  PROC DrawPart46()
    MoveL Offs(pOrigin,300.79,272.54,0.00),v40,fine,tPen\WObj:=wPaper;
    MoveL Offs(pOrigin,300.79,272.54,6.00),v60,z5,tPen\WObj:=wPaper;
    MoveL Offs(pOrigin,301.42,271.48,6.00),vTravel,z5,tPen\WObj:=wPaper;
    MoveL Offs(pOrigin,301.42,271.48,0.00),v60,z0,tPen\WObj:=wPaper;
    MoveL Offs(pOrigin,301.00,272.11,0.00),v40,z0,tPen\WObj:=wPaper;
    MoveL Offs(pOrigin,301.42,271.48,0.00),v40,z0,tPen\WObj:=wPaper;
    MoveL Offs(pOrigin,301.85,270.62,0.00),v40,z0,tPen\WObj:=wPaper;
    MoveL Offs(pOrigin,301.64,271.05,0.00),v40,z0,tPen\WObj:=wPaper;
    MoveL Offs(pOrigin,301.85,270.62,0.00),v40,fine,tPen\WObj:=wPaper;
    MoveL Offs(pOrigin,301.85,270.62,6.00),v60,z5,tPen\WObj:=wPaper;
    MoveL Offs(pOrigin,295.90,275.73,6.00),vTravel,z5,tPen\WObj:=wPaper;
    MoveL Offs(pOrigin,295.90,275.73,0.00),v60,z0,tPen\WObj:=wPaper;
    MoveL Offs(pOrigin,296.96,276.43,0.00),v40,z0,tPen\WObj:=wPaper;
    MoveL Offs(pOrigin,297.39,277.21,0.00),v40,z0,tPen\WObj:=wPaper;
    MoveL Offs(pOrigin,297.32,277.85,0.00),v40,z0,tPen\WObj:=wPaper;
    MoveL Offs(pOrigin,296.54,278.27,0.00),v40,z0,tPen\WObj:=wPaper;
    MoveL Offs(pOrigin,296.54,278.27,0.00),v40,z0,tPen\WObj:=wPaper;
    MoveL Offs(pOrigin,296.96,280.83,0.00),v40,z0,tPen\WObj:=wPaper;
    MoveL Offs(pOrigin,295.69,281.67,0.00),v40,z0,tPen\WObj:=wPaper;
    MoveL Offs(pOrigin,295.26,281.46,0.00),v40,z0,tPen\WObj:=wPaper;
    MoveL Offs(pOrigin,296.75,284.65,0.00),v40,fine,tPen\WObj:=wPaper;
    MoveL Offs(pOrigin,296.75,284.65,6.00),v60,z5,tPen\WObj:=wPaper;
    MoveL Offs(pOrigin,298.45,283.38,6.00),vTravel,z5,tPen\WObj:=wPaper;
    MoveL Offs(pOrigin,298.45,283.38,0.00),v60,z0,tPen\WObj:=wPaper;
    MoveL Offs(pOrigin,298.02,282.95,0.00),v40,z0,tPen\WObj:=wPaper;
    MoveL Offs(pOrigin,298.02,282.10,0.00),v40,z0,tPen\WObj:=wPaper;
    MoveL Offs(pOrigin,298.45,281.67,0.00),v40,z0,tPen\WObj:=wPaper;
    MoveL Offs(pOrigin,299.09,281.67,0.00),v40,fine,tPen\WObj:=wPaper;
    MoveL Offs(pOrigin,299.09,281.67,6.00),v60,z5,tPen\WObj:=wPaper;
    MoveL Offs(pOrigin,292.71,272.33,6.00),vTravel,z5,tPen\WObj:=wPaper;
    MoveL Offs(pOrigin,292.71,272.33,0.00),v60,z0,tPen\WObj:=wPaper;
    MoveL Offs(pOrigin,293.14,272.75,0.00),v40,z0,tPen\WObj:=wPaper;
    MoveL Offs(pOrigin,292.71,272.33,0.00),v40,fine,tPen\WObj:=wPaper;
    MoveL Offs(pOrigin,292.71,272.33,6.00),v60,z5,tPen\WObj:=wPaper;
    MoveL Offs(pOrigin,291.44,271.48,6.00),vTravel,z5,tPen\WObj:=wPaper;
    MoveL Offs(pOrigin,291.44,271.48,0.00),v60,z0,tPen\WObj:=wPaper;
    MoveL Offs(pOrigin,293.56,273.46,0.00),v40,z0,tPen\WObj:=wPaper;
    MoveL Offs(pOrigin,294.84,274.02,0.00),v40,z0,tPen\WObj:=wPaper;
    MoveL Offs(pOrigin,296.33,274.24,0.00),v40,z0,tPen\WObj:=wPaper;
    MoveL Offs(pOrigin,298.45,273.39,0.00),v40,z0,tPen\WObj:=wPaper;
    MoveL Offs(pOrigin,299.80,271.90,0.00),v40,z0,tPen\WObj:=wPaper;
    MoveL Offs(pOrigin,301.07,269.14,0.00),v40,z0,tPen\WObj:=wPaper;
    MoveL Offs(pOrigin,301.85,266.38,0.00),v40,z0,tPen\WObj:=wPaper;
    MoveL Offs(pOrigin,302.06,264.04,0.00),v40,z0,tPen\WObj:=wPaper;
    MoveL Offs(pOrigin,298.66,250.44,0.00),v40,z0,tPen\WObj:=wPaper;
    MoveL Offs(pOrigin,296.68,240.88,0.00),v40,z0,tPen\WObj:=wPaper;
    MoveL Offs(pOrigin,295.05,239.10,0.00),v40,z0,tPen\WObj:=wPaper;
    MoveL Offs(pOrigin,293.99,238.75,0.00),v40,z0,tPen\WObj:=wPaper;
    MoveL Offs(pOrigin,292.71,239.10,0.00),v40,z0,tPen\WObj:=wPaper;
    MoveL Offs(pOrigin,291.86,240.45,0.00),v40,z0,tPen\WObj:=wPaper;
    MoveL Offs(pOrigin,291.58,243.43,0.00),v40,z0,tPen\WObj:=wPaper;
    MoveL Offs(pOrigin,291.01,243.85,0.00),v40,fine,tPen\WObj:=wPaper;
    MoveL Offs(pOrigin,291.01,243.85,6.00),v60,z5,tPen\WObj:=wPaper;
    MoveL Offs(pOrigin,295.48,239.60,6.00),vTravel,z5,tPen\WObj:=wPaper;
    MoveL Offs(pOrigin,295.48,239.60,0.00),v60,z0,tPen\WObj:=wPaper;
    MoveL Offs(pOrigin,296.11,240.24,0.00),v40,z0,tPen\WObj:=wPaper;
    MoveL Offs(pOrigin,295.48,239.60,0.00),v40,fine,tPen\WObj:=wPaper;
    MoveL Offs(pOrigin,295.48,239.60,6.00),v60,z5,tPen\WObj:=wPaper;
    MoveL Offs(pOrigin,296.33,238.32,6.00),vTravel,z5,tPen\WObj:=wPaper;
    MoveL Offs(pOrigin,296.33,238.32,0.00),v60,z0,tPen\WObj:=wPaper;
    MoveL Offs(pOrigin,296.96,238.96,0.00),v40,z0,tPen\WObj:=wPaper;
    MoveL Offs(pOrigin,296.33,238.32,0.00),v40,fine,tPen\WObj:=wPaper;
    MoveL Offs(pOrigin,296.33,238.32,6.00),v60,z5,tPen\WObj:=wPaper;
    MoveL Offs(pOrigin,297.81,239.39,6.00),vTravel,z5,tPen\WObj:=wPaper;
    MoveL Offs(pOrigin,297.81,239.39,0.00),v60,z0,tPen\WObj:=wPaper;
    MoveL Offs(pOrigin,298.45,239.81,0.00),v40,z0,tPen\WObj:=wPaper;
    MoveL Offs(pOrigin,300.15,239.81,0.00),v40,z0,tPen\WObj:=wPaper;
    MoveL Offs(pOrigin,300.15,239.81,0.00),v40,z0,tPen\WObj:=wPaper;
    MoveL Offs(pOrigin,300.79,240.24,0.00),v40,z0,tPen\WObj:=wPaper;
    MoveL Offs(pOrigin,315.02,240.24,0.00),v40,z0,tPen\WObj:=wPaper;
    MoveL Offs(pOrigin,327.99,239.60,0.00),v40,z0,tPen\WObj:=wPaper;
    MoveL Offs(pOrigin,342.44,238.32,0.00),v40,z0,tPen\WObj:=wPaper;
    MoveL Offs(pOrigin,358.16,235.99,0.00),v40,z0,tPen\WObj:=wPaper;
    MoveL Offs(pOrigin,364.75,234.00,0.00),v40,z0,tPen\WObj:=wPaper;
    MoveL Offs(pOrigin,365.17,233.23,0.00),v40,z0,tPen\WObj:=wPaper;
    MoveL Offs(pOrigin,365.17,233.23,0.00),v40,z0,tPen\WObj:=wPaper;
    MoveL Offs(pOrigin,366.66,232.66,0.00),v40,z0,tPen\WObj:=wPaper;
    MoveL Offs(pOrigin,369.21,230.89,0.00),v40,z0,tPen\WObj:=wPaper;
    MoveL Offs(pOrigin,371.34,228.55,0.00),v40,z0,tPen\WObj:=wPaper;
    MoveL Offs(pOrigin,373.53,224.51,0.00),v40,z0,tPen\WObj:=wPaper;
    MoveL Offs(pOrigin,375.38,218.35,0.00),v40,z0,tPen\WObj:=wPaper;
    MoveL Offs(pOrigin,375.38,218.35,0.00),v40,z0,tPen\WObj:=wPaper;
    MoveL Offs(pOrigin,375.38,217.07,0.00),v40,z0,tPen\WObj:=wPaper;
    MoveL Offs(pOrigin,375.80,216.86,0.00),v40,z0,tPen\WObj:=wPaper;
    MoveL Offs(pOrigin,375.80,216.86,0.00),v40,z0,tPen\WObj:=wPaper;
    MoveL Offs(pOrigin,376.44,217.50,0.00),v40,z0,tPen\WObj:=wPaper;
    MoveL Offs(pOrigin,376.23,218.35,0.00),v40,z0,tPen\WObj:=wPaper;
    MoveL Offs(pOrigin,375.38,218.35,0.00),v40,z0,tPen\WObj:=wPaper;
    MoveL Offs(pOrigin,376.01,218.42,0.00),v40,z0,tPen\WObj:=wPaper;
    MoveL Offs(pOrigin,376.23,218.77,0.00),v40,z0,tPen\WObj:=wPaper;
    MoveL Offs(pOrigin,376.23,222.39,0.00),v40,z0,tPen\WObj:=wPaper;
    MoveL Offs(pOrigin,375.59,226.43,0.00),v40,z0,tPen\WObj:=wPaper;
    MoveL Offs(pOrigin,374.38,230.46,0.00),v40,z0,tPen\WObj:=wPaper;
    MoveL Offs(pOrigin,372.12,234.07,0.00),v40,z0,tPen\WObj:=wPaper;
    MoveL Offs(pOrigin,370.27,235.70,0.00),v40,z0,tPen\WObj:=wPaper;
    MoveL Offs(pOrigin,368.58,236.62,0.00),v40,z0,tPen\WObj:=wPaper;
    MoveL Offs(pOrigin,369.00,236.41,0.00),v40,z0,tPen\WObj:=wPaper;
    MoveL Offs(pOrigin,369.42,236.20,0.00),v40,z0,tPen\WObj:=wPaper;
    MoveL Offs(pOrigin,369.00,236.41,0.00),v40,z0,tPen\WObj:=wPaper;
    MoveL Offs(pOrigin,368.15,236.84,0.00),v40,z0,tPen\WObj:=wPaper;
    MoveL Offs(pOrigin,364.75,238.11,0.00),v40,z0,tPen\WObj:=wPaper;
    MoveL Offs(pOrigin,361.56,238.82,0.00),v40,z0,tPen\WObj:=wPaper;
    MoveL Offs(pOrigin,361.14,239.39,0.00),v40,fine,tPen\WObj:=wPaper;
    MoveL Offs(pOrigin,361.14,239.39,6.00),v60,z5,tPen\WObj:=wPaper;
    MoveL Offs(pOrigin,357.52,239.60,6.00),vTravel,z5,tPen\WObj:=wPaper;
    MoveL Offs(pOrigin,357.52,239.60,0.00),v60,z0,tPen\WObj:=wPaper;
    MoveL Offs(pOrigin,364.75,239.39,0.00),v40,z0,tPen\WObj:=wPaper;
    MoveL Offs(pOrigin,369.21,237.97,0.00),v40,z0,tPen\WObj:=wPaper;
    MoveL Offs(pOrigin,371.55,236.62,0.00),v40,z0,tPen\WObj:=wPaper;
    MoveL Offs(pOrigin,373.25,235.14,0.00),v40,z0,tPen\WObj:=wPaper;
    MoveL Offs(pOrigin,374.81,233.01,0.00),v40,z0,tPen\WObj:=wPaper;
    MoveL Offs(pOrigin,375.87,230.68,0.00),v40,z0,tPen\WObj:=wPaper;
    MoveL Offs(pOrigin,377.08,226.64,0.00),v40,z0,tPen\WObj:=wPaper;
    MoveL Offs(pOrigin,377.71,221.96,0.00),v40,z0,tPen\WObj:=wPaper;
    MoveL Offs(pOrigin,377.71,212.82,0.00),v40,z0,tPen\WObj:=wPaper;
    MoveL Offs(pOrigin,376.86,204.96,0.00),v40,z0,tPen\WObj:=wPaper;
    MoveL Offs(pOrigin,373.89,190.51,0.00),v40,z0,tPen\WObj:=wPaper;
    MoveL Offs(pOrigin,376.23,188.60,0.00),v40,z0,tPen\WObj:=wPaper;
    MoveL Offs(pOrigin,377.92,186.48,0.00),v40,z0,tPen\WObj:=wPaper;
    MoveL Offs(pOrigin,378.35,186.90,0.00),v40,z0,tPen\WObj:=wPaper;
  ENDPROC

  PROC DrawPart47()
    MoveL Offs(pOrigin,380.26,204.75,0.00),v40,z0,tPen\WObj:=wPaper;
    MoveL Offs(pOrigin,380.48,217.93,0.00),v40,z0,tPen\WObj:=wPaper;
    MoveL Offs(pOrigin,379.62,225.79,0.00),v40,z0,tPen\WObj:=wPaper;
    MoveL Offs(pOrigin,378.99,228.55,0.00),v40,z0,tPen\WObj:=wPaper;
    MoveL Offs(pOrigin,377.50,232.59,0.00),v40,z0,tPen\WObj:=wPaper;
    MoveL Offs(pOrigin,377.50,233.44,0.00),v40,z0,tPen\WObj:=wPaper;
    MoveL Offs(pOrigin,377.50,233.44,0.00),v40,z0,tPen\WObj:=wPaper;
    MoveL Offs(pOrigin,378.35,233.30,0.00),v40,z0,tPen\WObj:=wPaper;
    MoveL Offs(pOrigin,379.41,231.52,0.00),v40,z0,tPen\WObj:=wPaper;
    MoveL Offs(pOrigin,379.41,231.52,0.00),v40,z0,tPen\WObj:=wPaper;
    MoveL Offs(pOrigin,380.33,231.10,0.00),v40,z0,tPen\WObj:=wPaper;
    MoveL Offs(pOrigin,381.61,228.55,0.00),v40,z0,tPen\WObj:=wPaper;
    MoveL Offs(pOrigin,383.45,222.39,0.00),v40,z0,tPen\WObj:=wPaper;
    MoveL Offs(pOrigin,384.30,217.50,0.00),v40,z0,tPen\WObj:=wPaper;
    MoveL Offs(pOrigin,388.55,169.69,0.00),v40,z0,tPen\WObj:=wPaper;
    MoveL Offs(pOrigin,392.80,129.31,0.00),v40,z0,tPen\WObj:=wPaper;
    MoveL Offs(pOrigin,392.59,128.46,0.00),v40,z0,tPen\WObj:=wPaper;
    MoveL Offs(pOrigin,391.60,128.68,0.00),v40,z0,tPen\WObj:=wPaper;
    MoveL Offs(pOrigin,391.10,129.95,0.00),v40,z0,tPen\WObj:=wPaper;
    MoveL Offs(pOrigin,390.46,139.30,0.00),v40,z0,tPen\WObj:=wPaper;
    MoveL Offs(pOrigin,389.54,141.43,0.00),v40,z0,tPen\WObj:=wPaper;
    MoveL Offs(pOrigin,387.13,143.76,0.00),v40,z0,tPen\WObj:=wPaper;
    MoveL Offs(pOrigin,386.85,144.61,0.00),v40,z0,tPen\WObj:=wPaper;
    MoveL Offs(pOrigin,387.27,147.16,0.00),v40,z0,tPen\WObj:=wPaper;
    MoveL Offs(pOrigin,387.06,149.71,0.00),v40,z0,tPen\WObj:=wPaper;
    MoveL Offs(pOrigin,385.01,155.02,0.00),v40,z0,tPen\WObj:=wPaper;
    MoveL Offs(pOrigin,382.53,159.91,0.00),v40,z0,tPen\WObj:=wPaper;
    MoveL Offs(pOrigin,380.90,164.80,0.00),v40,z0,tPen\WObj:=wPaper;
    MoveL Offs(pOrigin,380.90,166.93,0.00),v40,z0,tPen\WObj:=wPaper;
    MoveL Offs(pOrigin,381.75,169.26,0.00),v40,z0,tPen\WObj:=wPaper;
    MoveL Offs(pOrigin,381.75,171.39,0.00),v40,z0,tPen\WObj:=wPaper;
    MoveL Offs(pOrigin,379.20,179.25,0.00),v40,z0,tPen\WObj:=wPaper;
    MoveL Offs(pOrigin,378.56,182.65,0.00),v40,z0,tPen\WObj:=wPaper;
    MoveL Offs(pOrigin,378.77,185.62,0.00),v40,z0,tPen\WObj:=wPaper;
    MoveL Offs(pOrigin,378.77,185.62,0.00),v40,z0,tPen\WObj:=wPaper;
    MoveL Offs(pOrigin,377.92,185.84,0.00),v40,z0,tPen\WObj:=wPaper;
    MoveL Offs(pOrigin,378.35,186.90,0.00),v40,z0,tPen\WObj:=wPaper;
    MoveL Offs(pOrigin,378.99,186.90,0.00),v40,z0,tPen\WObj:=wPaper;
    MoveL Offs(pOrigin,381.11,199.86,0.00),v40,z0,tPen\WObj:=wPaper;
    MoveL Offs(pOrigin,381.96,211.12,0.00),v40,z0,tPen\WObj:=wPaper;
    MoveL Offs(pOrigin,381.54,221.96,0.00),v40,z0,tPen\WObj:=wPaper;
    MoveL Offs(pOrigin,381.11,224.94,0.00),v40,z0,tPen\WObj:=wPaper;
    MoveL Offs(pOrigin,379.41,230.68,0.00),v40,z0,tPen\WObj:=wPaper;
    MoveL Offs(pOrigin,379.41,231.52,0.00),v40,fine,tPen\WObj:=wPaper;
    MoveL Offs(pOrigin,379.41,231.52,6.00),v60,z5,tPen\WObj:=wPaper;
    MoveL Offs(pOrigin,380.48,230.46,6.00),vTravel,z5,tPen\WObj:=wPaper;
    MoveL Offs(pOrigin,380.48,230.46,0.00),v60,z0,tPen\WObj:=wPaper;
    MoveL Offs(pOrigin,380.26,230.89,0.00),v40,z0,tPen\WObj:=wPaper;
    MoveL Offs(pOrigin,380.48,230.46,0.00),v40,fine,tPen\WObj:=wPaper;
    MoveL Offs(pOrigin,380.48,230.46,6.00),v60,z5,tPen\WObj:=wPaper;
    MoveL Offs(pOrigin,381.75,231.52,6.00),vTravel,z5,tPen\WObj:=wPaper;
    MoveL Offs(pOrigin,381.75,231.52,0.00),v60,z0,tPen\WObj:=wPaper;
    MoveL Offs(pOrigin,381.54,231.95,0.00),v40,z0,tPen\WObj:=wPaper;
    MoveL Offs(pOrigin,381.75,231.52,0.00),v40,fine,tPen\WObj:=wPaper;
    MoveL Offs(pOrigin,381.75,231.52,6.00),v60,z5,tPen\WObj:=wPaper;
    MoveL Offs(pOrigin,380.69,233.23,6.00),vTravel,z5,tPen\WObj:=wPaper;
    MoveL Offs(pOrigin,380.69,233.23,0.00),v60,z0,tPen\WObj:=wPaper;
    MoveL Offs(pOrigin,380.26,233.86,0.00),v40,z0,tPen\WObj:=wPaper;
    MoveL Offs(pOrigin,380.69,233.23,0.00),v40,fine,tPen\WObj:=wPaper;
    MoveL Offs(pOrigin,380.69,233.23,6.00),v60,z5,tPen\WObj:=wPaper;
    MoveL Offs(pOrigin,379.84,234.29,6.00),vTravel,z5,tPen\WObj:=wPaper;
    MoveL Offs(pOrigin,379.84,234.29,0.00),v60,z0,tPen\WObj:=wPaper;
    MoveL Offs(pOrigin,379.41,234.93,0.00),v40,z0,tPen\WObj:=wPaper;
    MoveL Offs(pOrigin,379.84,234.29,0.00),v40,z0,tPen\WObj:=wPaper;
    MoveL Offs(pOrigin,379.20,235.14,0.00),v40,z0,tPen\WObj:=wPaper;
    MoveL Offs(pOrigin,377.71,236.62,0.00),v40,z0,tPen\WObj:=wPaper;
    MoveL Offs(pOrigin,379.20,235.14,0.00),v40,fine,tPen\WObj:=wPaper;
    MoveL Offs(pOrigin,379.20,235.14,6.00),v60,z5,tPen\WObj:=wPaper;
    MoveL Offs(pOrigin,377.50,233.44,6.00),vTravel,z5,tPen\WObj:=wPaper;
    MoveL Offs(pOrigin,377.50,233.44,0.00),v60,z0,tPen\WObj:=wPaper;
    MoveL Offs(pOrigin,377.08,234.50,0.00),v40,z0,tPen\WObj:=wPaper;
    MoveL Offs(pOrigin,375.66,235.42,0.00),v40,z0,tPen\WObj:=wPaper;
    MoveL Offs(pOrigin,373.46,237.69,0.00),v40,z0,tPen\WObj:=wPaper;
    MoveL Offs(pOrigin,373.04,237.90,0.00),v40,z0,tPen\WObj:=wPaper;
    MoveL Offs(pOrigin,369.42,239.39,0.00),v40,z0,tPen\WObj:=wPaper;
    MoveL Offs(pOrigin,364.54,240.66,0.00),v40,z0,tPen\WObj:=wPaper;
    MoveL Offs(pOrigin,356.89,241.94,0.00),v40,z0,tPen\WObj:=wPaper;
    MoveL Offs(pOrigin,341.38,243.64,0.00),v40,z0,tPen\WObj:=wPaper;
    MoveL Offs(pOrigin,320.55,244.91,0.00),v40,z0,tPen\WObj:=wPaper;
    MoveL Offs(pOrigin,302.06,245.12,0.00),v40,z0,tPen\WObj:=wPaper;
    MoveL Offs(pOrigin,299.30,244.91,0.00),v40,z0,tPen\WObj:=wPaper;
    MoveL Offs(pOrigin,298.88,244.27,0.00),v40,z0,tPen\WObj:=wPaper;
    MoveL Offs(pOrigin,297.88,240.24,0.00),v40,z0,tPen\WObj:=wPaper;
    MoveL Offs(pOrigin,298.02,239.81,0.00),v40,z0,tPen\WObj:=wPaper;
    MoveL Offs(pOrigin,298.02,239.81,0.00),v40,z0,tPen\WObj:=wPaper;
    MoveL Offs(pOrigin,295.26,237.83,0.00),v40,z0,tPen\WObj:=wPaper;
    MoveL Offs(pOrigin,294.20,237.48,0.00),v40,z0,tPen\WObj:=wPaper;
    MoveL Offs(pOrigin,291.93,237.69,0.00),v40,z0,tPen\WObj:=wPaper;
    MoveL Offs(pOrigin,291.44,233.44,0.00),v40,z0,tPen\WObj:=wPaper;
    MoveL Offs(pOrigin,289.24,226.43,0.00),v40,z0,tPen\WObj:=wPaper;
    MoveL Offs(pOrigin,295.97,218.35,0.00),v40,z0,tPen\WObj:=wPaper;
    MoveL Offs(pOrigin,300.79,213.75,0.00),v40,z0,tPen\WObj:=wPaper;
    MoveL Offs(pOrigin,310.14,211.34,0.00),v40,z0,tPen\WObj:=wPaper;
    MoveL Offs(pOrigin,317.58,208.86,0.00),v40,z0,tPen\WObj:=wPaper;
    MoveL Offs(pOrigin,336.27,201.07,0.00),v40,z0,tPen\WObj:=wPaper;
    MoveL Offs(pOrigin,346.90,197.52,0.00),v40,z0,tPen\WObj:=wPaper;
    MoveL Offs(pOrigin,366.88,192.21,0.00),v40,z0,tPen\WObj:=wPaper;
    MoveL Offs(pOrigin,371.76,190.51,0.00),v40,z0,tPen\WObj:=wPaper;
    MoveL Offs(pOrigin,372.33,190.58,0.00),v40,z0,tPen\WObj:=wPaper;
    MoveL Offs(pOrigin,373.89,196.89,0.00),v40,z0,tPen\WObj:=wPaper;
    MoveL Offs(pOrigin,375.38,205.18,0.00),v40,z0,tPen\WObj:=wPaper;
    MoveL Offs(pOrigin,375.80,208.79,0.00),v40,z0,tPen\WObj:=wPaper;
    MoveL Offs(pOrigin,375.80,216.86,0.00),v40,fine,tPen\WObj:=wPaper;
    MoveL Offs(pOrigin,375.80,216.86,6.00),v60,z5,tPen\WObj:=wPaper;
    MoveL Offs(pOrigin,371.98,227.27,6.00),vTravel,z5,tPen\WObj:=wPaper;
    MoveL Offs(pOrigin,371.98,227.27,0.00),v60,z0,tPen\WObj:=wPaper;
    MoveL Offs(pOrigin,371.55,227.91,0.00),v40,z0,tPen\WObj:=wPaper;
    MoveL Offs(pOrigin,371.98,227.27,0.00),v40,fine,tPen\WObj:=wPaper;
    MoveL Offs(pOrigin,371.98,227.27,6.00),v60,z5,tPen\WObj:=wPaper;
    MoveL Offs(pOrigin,370.49,229.40,6.00),vTravel,z5,tPen\WObj:=wPaper;
    MoveL Offs(pOrigin,370.49,229.40,0.00),v60,z0,tPen\WObj:=wPaper;
    MoveL Offs(pOrigin,369.85,230.04,0.00),v40,z0,tPen\WObj:=wPaper;
    MoveL Offs(pOrigin,370.49,229.40,0.00),v40,fine,tPen\WObj:=wPaper;
    MoveL Offs(pOrigin,370.49,229.40,6.00),v60,z5,tPen\WObj:=wPaper;
    MoveL Offs(pOrigin,369.64,230.25,6.00),vTravel,z5,tPen\WObj:=wPaper;
    MoveL Offs(pOrigin,369.64,230.25,0.00),v60,z0,tPen\WObj:=wPaper;
    MoveL Offs(pOrigin,369.00,230.89,0.00),v40,z0,tPen\WObj:=wPaper;
    MoveL Offs(pOrigin,369.64,230.25,0.00),v40,fine,tPen\WObj:=wPaper;
    MoveL Offs(pOrigin,369.64,230.25,6.00),v60,z5,tPen\WObj:=wPaper;
    MoveL Offs(pOrigin,373.46,231.95,6.00),vTravel,z5,tPen\WObj:=wPaper;
  ENDPROC

  PROC DrawPart48()
    MoveL Offs(pOrigin,373.46,231.95,0.00),v60,z0,tPen\WObj:=wPaper;
    MoveL Offs(pOrigin,373.25,232.38,0.00),v40,z0,tPen\WObj:=wPaper;
    MoveL Offs(pOrigin,373.46,231.95,0.00),v40,fine,tPen\WObj:=wPaper;
    MoveL Offs(pOrigin,373.46,231.95,6.00),v60,z5,tPen\WObj:=wPaper;
    MoveL Offs(pOrigin,374.10,230.68,6.00),vTravel,z5,tPen\WObj:=wPaper;
    MoveL Offs(pOrigin,374.10,230.68,0.00),v60,z0,tPen\WObj:=wPaper;
    MoveL Offs(pOrigin,373.89,231.10,0.00),v40,z0,tPen\WObj:=wPaper;
    MoveL Offs(pOrigin,374.10,230.68,0.00),v40,fine,tPen\WObj:=wPaper;
    MoveL Offs(pOrigin,374.10,230.68,6.00),v60,z5,tPen\WObj:=wPaper;
    MoveL Offs(pOrigin,375.16,231.95,6.00),vTravel,z5,tPen\WObj:=wPaper;
    MoveL Offs(pOrigin,375.16,231.95,0.00),v60,z0,tPen\WObj:=wPaper;
    MoveL Offs(pOrigin,374.95,232.38,0.00),v40,z0,tPen\WObj:=wPaper;
    MoveL Offs(pOrigin,375.16,231.95,0.00),v40,z0,tPen\WObj:=wPaper;
    MoveL Offs(pOrigin,374.74,232.80,0.00),v40,z0,tPen\WObj:=wPaper;
    MoveL Offs(pOrigin,374.31,233.44,0.00),v40,z0,tPen\WObj:=wPaper;
    MoveL Offs(pOrigin,374.74,232.80,0.00),v40,fine,tPen\WObj:=wPaper;
    MoveL Offs(pOrigin,374.74,232.80,6.00),v60,z5,tPen\WObj:=wPaper;
    MoveL Offs(pOrigin,374.10,233.86,6.00),vTravel,z5,tPen\WObj:=wPaper;
    MoveL Offs(pOrigin,374.10,233.86,0.00),v60,z0,tPen\WObj:=wPaper;
    MoveL Offs(pOrigin,373.46,234.50,0.00),v40,z0,tPen\WObj:=wPaper;
    MoveL Offs(pOrigin,374.10,233.86,0.00),v40,fine,tPen\WObj:=wPaper;
    MoveL Offs(pOrigin,374.10,233.86,6.00),v60,z5,tPen\WObj:=wPaper;
    MoveL Offs(pOrigin,373.25,234.93,6.00),vTravel,z5,tPen\WObj:=wPaper;
    MoveL Offs(pOrigin,373.25,234.93,0.00),v60,z0,tPen\WObj:=wPaper;
    MoveL Offs(pOrigin,372.40,235.77,0.00),v40,z0,tPen\WObj:=wPaper;
    MoveL Offs(pOrigin,373.25,234.93,0.00),v40,fine,tPen\WObj:=wPaper;
    MoveL Offs(pOrigin,373.25,234.93,6.00),v60,z5,tPen\WObj:=wPaper;
    MoveL Offs(pOrigin,372.61,233.44,6.00),vTravel,z5,tPen\WObj:=wPaper;
    MoveL Offs(pOrigin,372.61,233.44,0.00),v60,z0,tPen\WObj:=wPaper;
    MoveL Offs(pOrigin,372.83,233.01,0.00),v40,z0,tPen\WObj:=wPaper;
    MoveL Offs(pOrigin,372.61,233.44,0.00),v40,z0,tPen\WObj:=wPaper;
    MoveL Offs(pOrigin,372.19,233.65,0.00),v40,z0,tPen\WObj:=wPaper;
    MoveL Offs(pOrigin,371.98,234.07,0.00),v40,z0,tPen\WObj:=wPaper;
    MoveL Offs(pOrigin,372.19,233.65,0.00),v40,fine,tPen\WObj:=wPaper;
    MoveL Offs(pOrigin,372.19,233.65,6.00),v60,z5,tPen\WObj:=wPaper;
    MoveL Offs(pOrigin,370.70,235.35,6.00),vTravel,z5,tPen\WObj:=wPaper;
    MoveL Offs(pOrigin,370.70,235.35,0.00),v60,z0,tPen\WObj:=wPaper;
    MoveL Offs(pOrigin,371.12,235.14,0.00),v40,z0,tPen\WObj:=wPaper;
    MoveL Offs(pOrigin,370.70,235.35,0.00),v40,z0,tPen\WObj:=wPaper;
    MoveL Offs(pOrigin,369.85,235.99,0.00),v40,z0,tPen\WObj:=wPaper;
    MoveL Offs(pOrigin,370.27,235.56,0.00),v40,z0,tPen\WObj:=wPaper;
    MoveL Offs(pOrigin,369.85,235.99,0.00),v40,fine,tPen\WObj:=wPaper;
    MoveL Offs(pOrigin,369.85,235.99,6.00),v60,z5,tPen\WObj:=wPaper;
    MoveL Offs(pOrigin,371.76,236.20,6.00),vTravel,z5,tPen\WObj:=wPaper;
    MoveL Offs(pOrigin,371.76,236.20,0.00),v60,z0,tPen\WObj:=wPaper;
    MoveL Offs(pOrigin,371.34,236.62,0.00),v40,z0,tPen\WObj:=wPaper;
    MoveL Offs(pOrigin,371.76,236.20,0.00),v40,fine,tPen\WObj:=wPaper;
    MoveL Offs(pOrigin,371.76,236.20,6.00),v60,z5,tPen\WObj:=wPaper;
    MoveL Offs(pOrigin,373.89,237.48,6.00),vTravel,z5,tPen\WObj:=wPaper;
    MoveL Offs(pOrigin,373.89,237.48,0.00),v60,z0,tPen\WObj:=wPaper;
    MoveL Offs(pOrigin,374.10,237.05,0.00),v40,z0,tPen\WObj:=wPaper;
    MoveL Offs(pOrigin,373.89,237.48,0.00),v40,z0,tPen\WObj:=wPaper;
    MoveL Offs(pOrigin,374.52,236.84,0.00),v40,z0,tPen\WObj:=wPaper;
    MoveL Offs(pOrigin,374.74,236.41,0.00),v40,z0,tPen\WObj:=wPaper;
    MoveL Offs(pOrigin,374.52,236.84,0.00),v40,z0,tPen\WObj:=wPaper;
    MoveL Offs(pOrigin,375.16,236.20,0.00),v40,z0,tPen\WObj:=wPaper;
    MoveL Offs(pOrigin,375.38,235.77,0.00),v40,z0,tPen\WObj:=wPaper;
    MoveL Offs(pOrigin,375.16,236.20,0.00),v40,fine,tPen\WObj:=wPaper;
    MoveL Offs(pOrigin,375.16,236.20,6.00),v60,z5,tPen\WObj:=wPaper;
    MoveL Offs(pOrigin,365.17,233.23,6.00),vTravel,z5,tPen\WObj:=wPaper;
    MoveL Offs(pOrigin,365.17,233.23,0.00),v60,z0,tPen\WObj:=wPaper;
    MoveL Offs(pOrigin,356.46,235.35,0.00),v40,z0,tPen\WObj:=wPaper;
    MoveL Offs(pOrigin,339.89,237.48,0.00),v40,z0,tPen\WObj:=wPaper;
    MoveL Offs(pOrigin,320.12,238.96,0.00),v40,z0,tPen\WObj:=wPaper;
    MoveL Offs(pOrigin,300.58,239.39,0.00),v40,z0,tPen\WObj:=wPaper;
    MoveL Offs(pOrigin,300.15,239.81,0.00),v40,fine,tPen\WObj:=wPaper;
    MoveL Offs(pOrigin,300.15,239.81,6.00),v60,z5,tPen\WObj:=wPaper;
    MoveL Offs(pOrigin,289.52,226.21,6.00),vTravel,z5,tPen\WObj:=wPaper;
    MoveL Offs(pOrigin,289.52,226.21,0.00),v60,z0,tPen\WObj:=wPaper;
    MoveL Offs(pOrigin,289.74,225.79,0.00),v40,z0,tPen\WObj:=wPaper;
    MoveL Offs(pOrigin,289.52,226.21,0.00),v40,fine,tPen\WObj:=wPaper;
    MoveL Offs(pOrigin,289.52,226.21,6.00),v60,z5,tPen\WObj:=wPaper;
    MoveL Offs(pOrigin,290.59,224.94,6.00),vTravel,z5,tPen\WObj:=wPaper;
    MoveL Offs(pOrigin,290.59,224.94,0.00),v60,z0,tPen\WObj:=wPaper;
    MoveL Offs(pOrigin,290.80,224.51,0.00),v40,z0,tPen\WObj:=wPaper;
    MoveL Offs(pOrigin,290.59,224.94,0.00),v40,fine,tPen\WObj:=wPaper;
    MoveL Offs(pOrigin,290.59,224.94,6.00),v60,z5,tPen\WObj:=wPaper;
    MoveL Offs(pOrigin,289.52,223.24,6.00),vTravel,z5,tPen\WObj:=wPaper;
    MoveL Offs(pOrigin,289.52,223.24,0.00),v60,z0,tPen\WObj:=wPaper;
    MoveL Offs(pOrigin,290.80,222.60,0.00),v40,z0,tPen\WObj:=wPaper;
    MoveL Offs(pOrigin,294.20,218.35,0.00),v40,z0,tPen\WObj:=wPaper;
    MoveL Offs(pOrigin,301.21,211.34,0.00),v40,z0,tPen\WObj:=wPaper;
    MoveL Offs(pOrigin,313.75,195.61,0.00),v40,z0,tPen\WObj:=wPaper;
    MoveL Offs(pOrigin,313.68,194.76,0.00),v40,z0,tPen\WObj:=wPaper;
    MoveL Offs(pOrigin,302.06,189.24,0.00),v40,z0,tPen\WObj:=wPaper;
    MoveL Offs(pOrigin,300.79,189.38,0.00),v40,z0,tPen\WObj:=wPaper;
    MoveL Offs(pOrigin,297.81,191.22,0.00),v40,z0,tPen\WObj:=wPaper;
    MoveL Offs(pOrigin,297.32,190.94,0.00),v40,z0,tPen\WObj:=wPaper;
    MoveL Offs(pOrigin,297.39,190.51,0.00),v40,z0,tPen\WObj:=wPaper;
    MoveL Offs(pOrigin,302.27,187.47,0.00),v40,z0,tPen\WObj:=wPaper;
    MoveL Offs(pOrigin,316.94,182.23,0.00),v40,z0,tPen\WObj:=wPaper;
    MoveL Offs(pOrigin,317.15,181.59,0.00),v40,z0,tPen\WObj:=wPaper;
    MoveL Offs(pOrigin,309.71,159.27,0.00),v40,z0,tPen\WObj:=wPaper;
    MoveL Offs(pOrigin,291.65,101.26,0.00),v40,z0,tPen\WObj:=wPaper;
    MoveL Offs(pOrigin,286.98,81.71,0.00),v40,z0,tPen\WObj:=wPaper;
    MoveL Offs(pOrigin,285.49,73.21,0.00),v40,z0,tPen\WObj:=wPaper;
    MoveL Offs(pOrigin,285.06,68.75,0.00),v40,z0,tPen\WObj:=wPaper;
    MoveL Offs(pOrigin,281.88,68.54,0.00),v40,z0,tPen\WObj:=wPaper;
    MoveL Offs(pOrigin,276.14,66.62,0.00),v40,z0,tPen\WObj:=wPaper;
    MoveL Offs(pOrigin,275.50,68.54,0.00),v40,z0,tPen\WObj:=wPaper;
    MoveL Offs(pOrigin,273.59,80.44,0.00),v40,z0,tPen\WObj:=wPaper;
    MoveL Offs(pOrigin,272.31,92.97,0.00),v40,z0,tPen\WObj:=wPaper;
    MoveL Offs(pOrigin,271.89,100.41,0.00),v40,z0,tPen\WObj:=wPaper;
    MoveL Offs(pOrigin,271.89,111.68,0.00),v40,z0,tPen\WObj:=wPaper;
    MoveL Offs(pOrigin,272.52,122.30,0.00),v40,z0,tPen\WObj:=wPaper;
    MoveL Offs(pOrigin,274.23,137.18,0.00),v40,z0,tPen\WObj:=wPaper;
    MoveL Offs(pOrigin,277.62,157.57,0.00),v40,z0,tPen\WObj:=wPaper;
    MoveL Offs(pOrigin,281.45,175.64,0.00),v40,z0,tPen\WObj:=wPaper;
    MoveL Offs(pOrigin,286.98,197.74,0.00),v40,z0,tPen\WObj:=wPaper;
    MoveL Offs(pOrigin,287.61,198.59,0.00),v40,fine,tPen\WObj:=wPaper;
    MoveL Offs(pOrigin,287.61,198.59,6.00),v60,z5,tPen\WObj:=wPaper;
    MoveL Offs(pOrigin,293.35,194.34,6.00),vTravel,z5,tPen\WObj:=wPaper;
    MoveL Offs(pOrigin,293.35,194.34,0.00),v60,z0,tPen\WObj:=wPaper;
    MoveL Offs(pOrigin,287.40,199.23,0.00),v40,z0,tPen\WObj:=wPaper;
    MoveL Offs(pOrigin,289.74,212.19,0.00),v40,z0,tPen\WObj:=wPaper;
    MoveL Offs(pOrigin,289.95,218.14,0.00),v40,z0,tPen\WObj:=wPaper;
    MoveL Offs(pOrigin,289.52,223.24,0.00),v40,fine,tPen\WObj:=wPaper;
    MoveL Offs(pOrigin,289.52,223.24,6.00),v60,z5,tPen\WObj:=wPaper;
    MoveL Offs(pOrigin,288.25,222.18,6.00),vTravel,z5,tPen\WObj:=wPaper;
    MoveL Offs(pOrigin,288.25,222.18,0.00),v60,z0,tPen\WObj:=wPaper;
  ENDPROC

  PROC DrawPart49()
    MoveL Offs(pOrigin,288.18,221.11,0.00),v40,z0,tPen\WObj:=wPaper;
    MoveL Offs(pOrigin,287.75,220.69,0.00),v40,z0,tPen\WObj:=wPaper;
    MoveL Offs(pOrigin,285.77,215.38,0.00),v40,z0,tPen\WObj:=wPaper;
    MoveL Offs(pOrigin,280.88,205.39,0.00),v40,z0,tPen\WObj:=wPaper;
    MoveL Offs(pOrigin,274.93,195.19,0.00),v40,z0,tPen\WObj:=wPaper;
    MoveL Offs(pOrigin,261.55,175.21,0.00),v40,z0,tPen\WObj:=wPaper;
    MoveL Offs(pOrigin,260.62,171.39,0.00),v40,z0,tPen\WObj:=wPaper;
    MoveL Offs(pOrigin,259.63,169.05,0.00),v40,z0,tPen\WObj:=wPaper;
    MoveL Offs(pOrigin,257.65,166.71,0.00),v40,z0,tPen\WObj:=wPaper;
    MoveL Offs(pOrigin,252.55,162.25,0.00),v40,z0,tPen\WObj:=wPaper;
    MoveL Offs(pOrigin,250.00,159.49,0.00),v40,z0,tPen\WObj:=wPaper;
    MoveL Offs(pOrigin,247.73,156.51,0.00),v40,z0,tPen\WObj:=wPaper;
    MoveL Offs(pOrigin,246.60,152.69,0.00),v40,z0,tPen\WObj:=wPaper;
    MoveL Offs(pOrigin,245.96,152.69,0.00),v40,z0,tPen\WObj:=wPaper;
    MoveL Offs(pOrigin,247.52,157.36,0.00),v40,z0,tPen\WObj:=wPaper;
    MoveL Offs(pOrigin,249.36,160.12,0.00),v40,z0,tPen\WObj:=wPaper;
    MoveL Offs(pOrigin,251.70,162.68,0.00),v40,z0,tPen\WObj:=wPaper;
    MoveL Offs(pOrigin,251.91,163.95,0.00),v40,z0,tPen\WObj:=wPaper;
    MoveL Offs(pOrigin,245.11,169.48,0.00),v40,z0,tPen\WObj:=wPaper;
    MoveL Offs(pOrigin,243.98,171.60,0.00),v40,z0,tPen\WObj:=wPaper;
    MoveL Offs(pOrigin,241.36,179.25,0.00),v40,z0,tPen\WObj:=wPaper;
    MoveL Offs(pOrigin,239.23,183.29,0.00),v40,z0,tPen\WObj:=wPaper;
    MoveL Offs(pOrigin,230.80,195.40,0.00),v40,z0,tPen\WObj:=wPaper;
    MoveL Offs(pOrigin,224.93,205.39,0.00),v40,z0,tPen\WObj:=wPaper;
    MoveL Offs(pOrigin,222.16,208.15,0.00),v40,z0,tPen\WObj:=wPaper;
    MoveL Offs(pOrigin,221.31,208.57,0.00),v40,z0,tPen\WObj:=wPaper;
    MoveL Offs(pOrigin,221.10,207.30,0.00),v40,z0,tPen\WObj:=wPaper;
    MoveL Offs(pOrigin,222.16,201.14,0.00),v40,z0,tPen\WObj:=wPaper;
    MoveL Offs(pOrigin,224.93,189.24,0.00),v40,z0,tPen\WObj:=wPaper;
    MoveL Offs(pOrigin,227.05,178.40,0.00),v40,z0,tPen\WObj:=wPaper;
    MoveL Offs(pOrigin,227.26,175.85,0.00),v40,z0,tPen\WObj:=wPaper;
    MoveL Offs(pOrigin,227.69,175.21,0.00),v40,z0,tPen\WObj:=wPaper;
    MoveL Offs(pOrigin,227.69,175.21,0.00),v40,z0,tPen\WObj:=wPaper;
    MoveL Offs(pOrigin,228.04,175.43,0.00),v40,z0,tPen\WObj:=wPaper;
    MoveL Offs(pOrigin,228.32,176.49,0.00),v40,z0,tPen\WObj:=wPaper;
    MoveL Offs(pOrigin,228.75,183.71,0.00),v40,z0,tPen\WObj:=wPaper;
    MoveL Offs(pOrigin,229.53,186.48,0.00),v40,z0,tPen\WObj:=wPaper;
    MoveL Offs(pOrigin,230.66,187.75,0.00),v40,z0,tPen\WObj:=wPaper;
    MoveL Offs(pOrigin,231.94,188.39,0.00),v40,z0,tPen\WObj:=wPaper;
    MoveL Offs(pOrigin,233.57,188.10,0.00),v40,z0,tPen\WObj:=wPaper;
    MoveL Offs(pOrigin,233.85,187.32,0.00),v40,z0,tPen\WObj:=wPaper;
    MoveL Offs(pOrigin,233.85,187.32,0.00),v40,z0,tPen\WObj:=wPaper;
    MoveL Offs(pOrigin,236.19,184.99,0.00),v40,z0,tPen\WObj:=wPaper;
    MoveL Offs(pOrigin,237.18,183.50,0.00),v40,z0,tPen\WObj:=wPaper;
    MoveL Offs(pOrigin,237.46,182.23,0.00),v40,z0,tPen\WObj:=wPaper;
    MoveL Offs(pOrigin,237.46,182.23,0.00),v40,z0,tPen\WObj:=wPaper;
    MoveL Offs(pOrigin,238.95,179.25,0.00),v40,z0,tPen\WObj:=wPaper;
    MoveL Offs(pOrigin,238.88,177.55,0.00),v40,z0,tPen\WObj:=wPaper;
    MoveL Offs(pOrigin,238.10,176.91,0.00),v40,z0,tPen\WObj:=wPaper;
    MoveL Offs(pOrigin,237.04,177.05,0.00),v40,z0,tPen\WObj:=wPaper;
    MoveL Offs(pOrigin,236.19,177.76,0.00),v40,z0,tPen\WObj:=wPaper;
    MoveL Offs(pOrigin,235.98,178.61,0.00),v40,z0,tPen\WObj:=wPaper;
    MoveL Offs(pOrigin,235.98,178.61,0.00),v40,z0,tPen\WObj:=wPaper;
    MoveL Offs(pOrigin,235.48,179.04,0.00),v40,z0,tPen\WObj:=wPaper;
    MoveL Offs(pOrigin,235.12,180.10,0.00),v40,z0,tPen\WObj:=wPaper;
    MoveL Offs(pOrigin,235.27,181.59,0.00),v40,z0,tPen\WObj:=wPaper;
    MoveL Offs(pOrigin,236.19,182.23,0.00),v40,z0,tPen\WObj:=wPaper;
    MoveL Offs(pOrigin,237.46,182.23,0.00),v40,fine,tPen\WObj:=wPaper;
    MoveL Offs(pOrigin,237.46,182.23,6.00),v60,z5,tPen\WObj:=wPaper;
    MoveL Offs(pOrigin,239.16,183.07,6.00),vTravel,z5,tPen\WObj:=wPaper;
    MoveL Offs(pOrigin,239.16,183.07,0.00),v60,z0,tPen\WObj:=wPaper;
    MoveL Offs(pOrigin,238.74,183.71,0.00),v40,z0,tPen\WObj:=wPaper;
    MoveL Offs(pOrigin,239.16,183.07,0.00),v40,fine,tPen\WObj:=wPaper;
    MoveL Offs(pOrigin,239.16,183.07,6.00),v60,z5,tPen\WObj:=wPaper;
    MoveL Offs(pOrigin,239.80,182.01,6.00),vTravel,z5,tPen\WObj:=wPaper;
    MoveL Offs(pOrigin,239.80,182.01,0.00),v60,z0,tPen\WObj:=wPaper;
    MoveL Offs(pOrigin,239.38,182.65,0.00),v40,z0,tPen\WObj:=wPaper;
    MoveL Offs(pOrigin,239.80,182.01,0.00),v40,fine,tPen\WObj:=wPaper;
    MoveL Offs(pOrigin,239.80,182.01,6.00),v60,z5,tPen\WObj:=wPaper;
    MoveL Offs(pOrigin,240.65,182.86,6.00),vTravel,z5,tPen\WObj:=wPaper;
    MoveL Offs(pOrigin,240.65,182.86,0.00),v60,z0,tPen\WObj:=wPaper;
    MoveL Offs(pOrigin,240.44,183.29,0.00),v40,z0,tPen\WObj:=wPaper;
    MoveL Offs(pOrigin,240.65,182.86,0.00),v40,fine,tPen\WObj:=wPaper;
    MoveL Offs(pOrigin,240.65,182.86,6.00),v60,z5,tPen\WObj:=wPaper;
    MoveL Offs(pOrigin,241.29,181.80,6.00),vTravel,z5,tPen\WObj:=wPaper;
    MoveL Offs(pOrigin,241.29,181.80,0.00),v60,z0,tPen\WObj:=wPaper;
    MoveL Offs(pOrigin,240.86,182.44,0.00),v40,z0,tPen\WObj:=wPaper;
    MoveL Offs(pOrigin,241.29,181.80,0.00),v40,fine,tPen\WObj:=wPaper;
    MoveL Offs(pOrigin,241.29,181.80,6.00),v60,z5,tPen\WObj:=wPaper;
    MoveL Offs(pOrigin,240.44,180.74,6.00),vTravel,z5,tPen\WObj:=wPaper;
    MoveL Offs(pOrigin,240.44,180.74,0.00),v60,z0,tPen\WObj:=wPaper;
    MoveL Offs(pOrigin,240.23,181.16,0.00),v40,z0,tPen\WObj:=wPaper;
    MoveL Offs(pOrigin,240.44,180.74,0.00),v40,fine,tPen\WObj:=wPaper;
    MoveL Offs(pOrigin,240.44,180.74,6.00),v60,z5,tPen\WObj:=wPaper;
    MoveL Offs(pOrigin,241.29,179.04,6.00),vTravel,z5,tPen\WObj:=wPaper;
    MoveL Offs(pOrigin,241.29,179.04,0.00),v60,z0,tPen\WObj:=wPaper;
    MoveL Offs(pOrigin,241.07,179.46,0.00),v40,z0,tPen\WObj:=wPaper;
    MoveL Offs(pOrigin,241.29,179.04,0.00),v40,fine,tPen\WObj:=wPaper;
    MoveL Offs(pOrigin,241.29,179.04,6.00),v60,z5,tPen\WObj:=wPaper;
    MoveL Offs(pOrigin,242.35,180.52,6.00),vTravel,z5,tPen\WObj:=wPaper;
    MoveL Offs(pOrigin,242.35,180.52,0.00),v60,z0,tPen\WObj:=wPaper;
    MoveL Offs(pOrigin,245.25,171.60,0.00),v40,z0,tPen\WObj:=wPaper;
    MoveL Offs(pOrigin,245.96,170.32,0.00),v40,z0,tPen\WObj:=wPaper;
    MoveL Offs(pOrigin,248.80,167.85,0.00),v40,z0,tPen\WObj:=wPaper;
    MoveL Offs(pOrigin,248.30,168.20,0.00),v40,z0,tPen\WObj:=wPaper;
    MoveL Offs(pOrigin,247.88,168.41,0.00),v40,z0,tPen\WObj:=wPaper;
    MoveL Offs(pOrigin,247.45,168.84,0.00),v40,z0,tPen\WObj:=wPaper;
    MoveL Offs(pOrigin,247.88,168.41,0.00),v40,fine,tPen\WObj:=wPaper;
    MoveL Offs(pOrigin,247.88,168.41,6.00),v60,z5,tPen\WObj:=wPaper;
    MoveL Offs(pOrigin,246.81,169.26,6.00),vTravel,z5,tPen\WObj:=wPaper;
    MoveL Offs(pOrigin,246.81,169.26,0.00),v60,z0,tPen\WObj:=wPaper;
    MoveL Offs(pOrigin,245.75,170.32,0.00),v40,z0,tPen\WObj:=wPaper;
    MoveL Offs(pOrigin,246.81,169.26,0.00),v40,fine,tPen\WObj:=wPaper;
    MoveL Offs(pOrigin,246.81,169.26,6.00),v60,z5,tPen\WObj:=wPaper;
    MoveL Offs(pOrigin,245.96,168.41,6.00),vTravel,z5,tPen\WObj:=wPaper;
    MoveL Offs(pOrigin,245.96,168.41,0.00),v60,z0,tPen\WObj:=wPaper;
    MoveL Offs(pOrigin,245.32,169.05,0.00),v40,z0,tPen\WObj:=wPaper;
    MoveL Offs(pOrigin,245.96,168.41,0.00),v40,fine,tPen\WObj:=wPaper;
    MoveL Offs(pOrigin,245.96,168.41,6.00),v60,z5,tPen\WObj:=wPaper;
    MoveL Offs(pOrigin,244.69,169.90,6.00),vTravel,z5,tPen\WObj:=wPaper;
    MoveL Offs(pOrigin,244.69,169.90,0.00),v60,z0,tPen\WObj:=wPaper;
    MoveL Offs(pOrigin,244.26,170.54,0.00),v40,z0,tPen\WObj:=wPaper;
    MoveL Offs(pOrigin,244.69,169.90,0.00),v40,fine,tPen\WObj:=wPaper;
    MoveL Offs(pOrigin,244.69,169.90,6.00),v60,z5,tPen\WObj:=wPaper;
    MoveL Offs(pOrigin,245.54,170.75,6.00),vTravel,z5,tPen\WObj:=wPaper;
    MoveL Offs(pOrigin,245.54,170.75,0.00),v60,z0,tPen\WObj:=wPaper;
    MoveL Offs(pOrigin,245.32,171.18,0.00),v40,z0,tPen\WObj:=wPaper;
    MoveL Offs(pOrigin,245.54,170.75,0.00),v40,fine,tPen\WObj:=wPaper;
    MoveL Offs(pOrigin,245.54,170.75,6.00),v60,z5,tPen\WObj:=wPaper;
    MoveL Offs(pOrigin,249.36,167.56,6.00),vTravel,z5,tPen\WObj:=wPaper;
  ENDPROC

  PROC DrawPart50()
    MoveL Offs(pOrigin,249.36,167.56,0.00),v60,z0,tPen\WObj:=wPaper;
    MoveL Offs(pOrigin,252.76,164.66,0.00),v40,z0,tPen\WObj:=wPaper;
    MoveL Offs(pOrigin,253.40,164.59,0.00),v40,z0,tPen\WObj:=wPaper;
    MoveL Offs(pOrigin,258.08,168.84,0.00),v40,z0,tPen\WObj:=wPaper;
    MoveL Offs(pOrigin,259.00,170.32,0.00),v40,z0,tPen\WObj:=wPaper;
    MoveL Offs(pOrigin,259.77,173.94,0.00),v40,z0,tPen\WObj:=wPaper;
    MoveL Offs(pOrigin,260.98,176.49,0.00),v40,z0,tPen\WObj:=wPaper;
    MoveL Offs(pOrigin,261.12,177.55,0.00),v40,z0,tPen\WObj:=wPaper;
    MoveL Offs(pOrigin,263.39,180.10,0.00),v40,z0,tPen\WObj:=wPaper;
    MoveL Offs(pOrigin,267.85,186.48,0.00),v40,z0,tPen\WObj:=wPaper;
    MoveL Offs(pOrigin,268.27,188.18,0.00),v40,z0,tPen\WObj:=wPaper;
    MoveL Offs(pOrigin,268.27,188.18,0.00),v40,z0,tPen\WObj:=wPaper;
    MoveL Offs(pOrigin,269.34,189.88,0.00),v40,z0,tPen\WObj:=wPaper;
    MoveL Offs(pOrigin,271.04,191.57,0.00),v40,z0,tPen\WObj:=wPaper;
    MoveL Offs(pOrigin,273.73,195.61,0.00),v40,z0,tPen\WObj:=wPaper;
    MoveL Offs(pOrigin,273.80,196.68,0.00),v40,fine,tPen\WObj:=wPaper;
    MoveL Offs(pOrigin,273.80,196.68,6.00),v60,z5,tPen\WObj:=wPaper;
    MoveL Offs(pOrigin,275.71,196.25,6.00),vTravel,z5,tPen\WObj:=wPaper;
    MoveL Offs(pOrigin,275.71,196.25,0.00),v60,z0,tPen\WObj:=wPaper;
    MoveL Offs(pOrigin,276.14,196.89,0.00),v40,z0,tPen\WObj:=wPaper;
    MoveL Offs(pOrigin,275.71,196.25,0.00),v40,fine,tPen\WObj:=wPaper;
    MoveL Offs(pOrigin,275.71,196.25,6.00),v60,z5,tPen\WObj:=wPaper;
    MoveL Offs(pOrigin,274.86,194.76,6.00),vTravel,z5,tPen\WObj:=wPaper;
    MoveL Offs(pOrigin,274.86,194.76,0.00),v60,z0,tPen\WObj:=wPaper;
    MoveL Offs(pOrigin,275.08,195.19,0.00),v40,z0,tPen\WObj:=wPaper;
    MoveL Offs(pOrigin,274.86,194.76,0.00),v40,fine,tPen\WObj:=wPaper;
    MoveL Offs(pOrigin,274.86,194.76,6.00),v60,z5,tPen\WObj:=wPaper;
    MoveL Offs(pOrigin,274.01,193.49,6.00),vTravel,z5,tPen\WObj:=wPaper;
    MoveL Offs(pOrigin,274.01,193.49,0.00),v60,z0,tPen\WObj:=wPaper;
    MoveL Offs(pOrigin,274.44,194.12,0.00),v40,z0,tPen\WObj:=wPaper;
    MoveL Offs(pOrigin,274.01,193.49,0.00),v40,z0,tPen\WObj:=wPaper;
    MoveL Offs(pOrigin,273.59,192.85,0.00),v40,z0,tPen\WObj:=wPaper;
    MoveL Offs(pOrigin,273.80,193.27,0.00),v40,z0,tPen\WObj:=wPaper;
    MoveL Offs(pOrigin,273.59,192.85,0.00),v40,fine,tPen\WObj:=wPaper;
    MoveL Offs(pOrigin,273.59,192.85,6.00),v60,z5,tPen\WObj:=wPaper;
    MoveL Offs(pOrigin,272.95,194.12,6.00),vTravel,z5,tPen\WObj:=wPaper;
    MoveL Offs(pOrigin,272.95,194.12,0.00),v60,z0,tPen\WObj:=wPaper;
    MoveL Offs(pOrigin,273.38,194.76,0.00),v40,z0,tPen\WObj:=wPaper;
    MoveL Offs(pOrigin,272.95,194.12,0.00),v40,fine,tPen\WObj:=wPaper;
    MoveL Offs(pOrigin,272.95,194.12,6.00),v60,z5,tPen\WObj:=wPaper;
    MoveL Offs(pOrigin,275.29,198.80,6.00),vTravel,z5,tPen\WObj:=wPaper;
    MoveL Offs(pOrigin,275.29,198.80,0.00),v60,z0,tPen\WObj:=wPaper;
    MoveL Offs(pOrigin,276.14,199.65,0.00),v40,z0,tPen\WObj:=wPaper;
    MoveL Offs(pOrigin,275.29,198.80,0.00),v40,fine,tPen\WObj:=wPaper;
    MoveL Offs(pOrigin,275.29,198.80,6.00),v60,z5,tPen\WObj:=wPaper;
    MoveL Offs(pOrigin,277.41,199.01,6.00),vTravel,z5,tPen\WObj:=wPaper;
    MoveL Offs(pOrigin,277.41,199.01,0.00),v60,z0,tPen\WObj:=wPaper;
    MoveL Offs(pOrigin,277.62,199.44,0.00),v40,z0,tPen\WObj:=wPaper;
    MoveL Offs(pOrigin,277.41,199.01,0.00),v40,z0,tPen\WObj:=wPaper;
    MoveL Offs(pOrigin,277.84,199.65,0.00),v40,z0,tPen\WObj:=wPaper;
    MoveL Offs(pOrigin,278.05,200.07,0.00),v40,z0,tPen\WObj:=wPaper;
    MoveL Offs(pOrigin,277.84,199.65,0.00),v40,fine,tPen\WObj:=wPaper;
    MoveL Offs(pOrigin,277.84,199.65,6.00),v60,z5,tPen\WObj:=wPaper;
    MoveL Offs(pOrigin,279.11,201.99,6.00),vTravel,z5,tPen\WObj:=wPaper;
    MoveL Offs(pOrigin,279.11,201.99,0.00),v60,z0,tPen\WObj:=wPaper;
    MoveL Offs(pOrigin,279.54,202.62,0.00),v40,z0,tPen\WObj:=wPaper;
    MoveL Offs(pOrigin,279.11,201.99,0.00),v40,fine,tPen\WObj:=wPaper;
    MoveL Offs(pOrigin,279.11,201.99,6.00),v60,z5,tPen\WObj:=wPaper;
    MoveL Offs(pOrigin,278.05,202.62,6.00),vTravel,z5,tPen\WObj:=wPaper;
    MoveL Offs(pOrigin,278.05,202.62,0.00),v60,z0,tPen\WObj:=wPaper;
    MoveL Offs(pOrigin,278.26,203.05,0.00),v40,z0,tPen\WObj:=wPaper;
    MoveL Offs(pOrigin,278.05,202.62,0.00),v40,fine,tPen\WObj:=wPaper;
    MoveL Offs(pOrigin,278.05,202.62,6.00),v60,z5,tPen\WObj:=wPaper;
    MoveL Offs(pOrigin,278.48,204.96,6.00),vTravel,z5,tPen\WObj:=wPaper;
    MoveL Offs(pOrigin,278.48,204.96,0.00),v60,z0,tPen\WObj:=wPaper;
    MoveL Offs(pOrigin,278.48,203.90,0.00),v40,z0,tPen\WObj:=wPaper;
    MoveL Offs(pOrigin,277.91,202.62,0.00),v40,z0,tPen\WObj:=wPaper;
    MoveL Offs(pOrigin,273.80,196.89,0.00),v40,z0,tPen\WObj:=wPaper;
    MoveL Offs(pOrigin,265.73,192.57,0.00),v40,z0,tPen\WObj:=wPaper;
    MoveL Offs(pOrigin,259.56,190.94,0.00),v40,z0,tPen\WObj:=wPaper;
    MoveL Offs(pOrigin,257.01,190.94,0.00),v40,z0,tPen\WObj:=wPaper;
    MoveL Offs(pOrigin,251.06,192.21,0.00),v40,z0,tPen\WObj:=wPaper;
    MoveL Offs(pOrigin,246.18,191.15,0.00),v40,z0,tPen\WObj:=wPaper;
    MoveL Offs(pOrigin,243.62,190.94,0.00),v40,z0,tPen\WObj:=wPaper;
    MoveL Offs(pOrigin,238.31,192.35,0.00),v40,z0,tPen\WObj:=wPaper;
    MoveL Offs(pOrigin,233.21,194.98,0.00),v40,z0,tPen\WObj:=wPaper;
    MoveL Offs(pOrigin,232.36,196.68,0.00),v40,z0,tPen\WObj:=wPaper;
    MoveL Offs(pOrigin,230.24,199.01,0.00),v40,z0,tPen\WObj:=wPaper;
    MoveL Offs(pOrigin,228.40,201.77,0.00),v40,z0,tPen\WObj:=wPaper;
    MoveL Offs(pOrigin,228.54,202.34,0.00),v40,z0,tPen\WObj:=wPaper;
    MoveL Offs(pOrigin,229.39,202.62,0.00),v40,fine,tPen\WObj:=wPaper;
    MoveL Offs(pOrigin,229.39,202.62,6.00),v60,z5,tPen\WObj:=wPaper;
    MoveL Offs(pOrigin,227.90,204.11,6.00),vTravel,z5,tPen\WObj:=wPaper;
    MoveL Offs(pOrigin,227.90,204.11,0.00),v60,z0,tPen\WObj:=wPaper;
    MoveL Offs(pOrigin,227.05,204.96,0.00),v40,z0,tPen\WObj:=wPaper;
    MoveL Offs(pOrigin,227.90,204.11,0.00),v40,fine,tPen\WObj:=wPaper;
    MoveL Offs(pOrigin,227.90,204.11,6.00),v60,z5,tPen\WObj:=wPaper;
    MoveL Offs(pOrigin,229.60,199.65,6.00),vTravel,z5,tPen\WObj:=wPaper;
    MoveL Offs(pOrigin,229.60,199.65,0.00),v60,z0,tPen\WObj:=wPaper;
    MoveL Offs(pOrigin,229.18,200.29,0.00),v40,z0,tPen\WObj:=wPaper;
    MoveL Offs(pOrigin,229.60,199.65,0.00),v40,fine,tPen\WObj:=wPaper;
    MoveL Offs(pOrigin,229.60,199.65,6.00),v60,z5,tPen\WObj:=wPaper;
    MoveL Offs(pOrigin,228.75,198.59,6.00),vTravel,z5,tPen\WObj:=wPaper;
    MoveL Offs(pOrigin,228.75,198.59,0.00),v60,z0,tPen\WObj:=wPaper;
    MoveL Offs(pOrigin,228.32,199.23,0.00),v40,z0,tPen\WObj:=wPaper;
    MoveL Offs(pOrigin,228.75,198.59,0.00),v40,fine,tPen\WObj:=wPaper;
    MoveL Offs(pOrigin,228.75,198.59,6.00),v60,z5,tPen\WObj:=wPaper;
    MoveL Offs(pOrigin,229.39,197.52,6.00),vTravel,z5,tPen\WObj:=wPaper;
    MoveL Offs(pOrigin,229.39,197.52,0.00),v60,z0,tPen\WObj:=wPaper;
    MoveL Offs(pOrigin,228.96,198.16,0.00),v40,z0,tPen\WObj:=wPaper;
    MoveL Offs(pOrigin,229.39,197.52,0.00),v40,fine,tPen\WObj:=wPaper;
    MoveL Offs(pOrigin,229.39,197.52,6.00),v60,z5,tPen\WObj:=wPaper;
    MoveL Offs(pOrigin,231.09,197.95,6.00),vTravel,z5,tPen\WObj:=wPaper;
    MoveL Offs(pOrigin,231.09,197.95,0.00),v60,z0,tPen\WObj:=wPaper;
    MoveL Offs(pOrigin,230.02,199.01,0.00),v40,z0,tPen\WObj:=wPaper;
    MoveL Offs(pOrigin,231.09,197.95,0.00),v40,z0,tPen\WObj:=wPaper;
    MoveL Offs(pOrigin,231.73,197.10,0.00),v40,z0,tPen\WObj:=wPaper;
    MoveL Offs(pOrigin,231.30,197.52,0.00),v40,z0,tPen\WObj:=wPaper;
    MoveL Offs(pOrigin,231.73,197.10,0.00),v40,fine,tPen\WObj:=wPaper;
    MoveL Offs(pOrigin,231.73,197.10,6.00),v60,z5,tPen\WObj:=wPaper;
    MoveL Offs(pOrigin,230.88,194.98,6.00),vTravel,z5,tPen\WObj:=wPaper;
    MoveL Offs(pOrigin,230.88,194.98,0.00),v60,z0,tPen\WObj:=wPaper;
    MoveL Offs(pOrigin,230.66,195.40,0.00),v40,z0,tPen\WObj:=wPaper;
    MoveL Offs(pOrigin,230.88,194.98,0.00),v40,fine,tPen\WObj:=wPaper;
    MoveL Offs(pOrigin,230.88,194.98,6.00),v60,z5,tPen\WObj:=wPaper;
    MoveL Offs(pOrigin,232.15,193.06,6.00),vTravel,z5,tPen\WObj:=wPaper;
    MoveL Offs(pOrigin,232.15,193.06,0.00),v60,z0,tPen\WObj:=wPaper;
    MoveL Offs(pOrigin,231.73,193.70,0.00),v40,z0,tPen\WObj:=wPaper;
    MoveL Offs(pOrigin,232.15,193.06,0.00),v40,fine,tPen\WObj:=wPaper;
    MoveL Offs(pOrigin,232.15,193.06,6.00),v60,z5,tPen\WObj:=wPaper;
  ENDPROC

  PROC DrawPart51()
    MoveL Offs(pOrigin,233.43,194.55,6.00),vTravel,z5,tPen\WObj:=wPaper;
    MoveL Offs(pOrigin,233.43,194.55,0.00),v60,z0,tPen\WObj:=wPaper;
    MoveL Offs(pOrigin,233.57,193.49,0.00),v40,z0,tPen\WObj:=wPaper;
    MoveL Offs(pOrigin,235.98,190.09,0.00),v40,z0,tPen\WObj:=wPaper;
    MoveL Offs(pOrigin,237.46,188.39,0.00),v40,z0,tPen\WObj:=wPaper;
    MoveL Offs(pOrigin,239.09,187.25,0.00),v40,z0,tPen\WObj:=wPaper;
    MoveL Offs(pOrigin,239.59,186.33,0.00),v40,z0,tPen\WObj:=wPaper;
    MoveL Offs(pOrigin,244.90,184.35,0.00),v40,z0,tPen\WObj:=wPaper;
    MoveL Offs(pOrigin,247.88,183.71,0.00),v40,z0,tPen\WObj:=wPaper;
    MoveL Offs(pOrigin,248.73,183.93,0.00),v40,fine,tPen\WObj:=wPaper;
    MoveL Offs(pOrigin,248.73,183.93,6.00),v60,z5,tPen\WObj:=wPaper;
    MoveL Offs(pOrigin,247.24,179.04,6.00),vTravel,z5,tPen\WObj:=wPaper;
    MoveL Offs(pOrigin,247.24,179.04,0.00),v60,z0,tPen\WObj:=wPaper;
    MoveL Offs(pOrigin,245.54,179.39,0.00),v40,z0,tPen\WObj:=wPaper;
    MoveL Offs(pOrigin,242.35,180.74,0.00),v40,z0,tPen\WObj:=wPaper;
    MoveL Offs(pOrigin,239.30,185.41,0.00),v40,z0,tPen\WObj:=wPaper;
    MoveL Offs(pOrigin,239.38,186.26,0.00),v40,fine,tPen\WObj:=wPaper;
    MoveL Offs(pOrigin,239.38,186.26,6.00),v60,z5,tPen\WObj:=wPaper;
    MoveL Offs(pOrigin,238.10,184.77,6.00),vTravel,z5,tPen\WObj:=wPaper;
    MoveL Offs(pOrigin,238.10,184.77,0.00),v60,z0,tPen\WObj:=wPaper;
    MoveL Offs(pOrigin,237.68,185.41,0.00),v40,z0,tPen\WObj:=wPaper;
    MoveL Offs(pOrigin,238.10,184.77,0.00),v40,fine,tPen\WObj:=wPaper;
    MoveL Offs(pOrigin,238.10,184.77,6.00),v60,z5,tPen\WObj:=wPaper;
    MoveL Offs(pOrigin,236.82,186.69,6.00),vTravel,z5,tPen\WObj:=wPaper;
    MoveL Offs(pOrigin,236.82,186.69,0.00),v60,z0,tPen\WObj:=wPaper;
    MoveL Offs(pOrigin,235.98,187.75,0.00),v40,z0,tPen\WObj:=wPaper;
    MoveL Offs(pOrigin,236.82,186.69,0.00),v40,fine,tPen\WObj:=wPaper;
    MoveL Offs(pOrigin,236.82,186.69,6.00),v60,z5,tPen\WObj:=wPaper;
    MoveL Offs(pOrigin,237.04,188.60,6.00),vTravel,z5,tPen\WObj:=wPaper;
    MoveL Offs(pOrigin,237.04,188.60,0.00),v60,z0,tPen\WObj:=wPaper;
    MoveL Offs(pOrigin,236.40,189.24,0.00),v40,z0,tPen\WObj:=wPaper;
    MoveL Offs(pOrigin,237.04,188.60,0.00),v40,fine,tPen\WObj:=wPaper;
    MoveL Offs(pOrigin,237.04,188.60,6.00),v60,z5,tPen\WObj:=wPaper;
    MoveL Offs(pOrigin,235.76,190.09,6.00),vTravel,z5,tPen\WObj:=wPaper;
    MoveL Offs(pOrigin,235.76,190.09,0.00),v60,z0,tPen\WObj:=wPaper;
    MoveL Offs(pOrigin,235.34,190.73,0.00),v40,z0,tPen\WObj:=wPaper;
    MoveL Offs(pOrigin,235.76,190.09,0.00),v40,fine,tPen\WObj:=wPaper;
    MoveL Offs(pOrigin,235.76,190.09,6.00),v60,z5,tPen\WObj:=wPaper;
    MoveL Offs(pOrigin,235.12,191.15,6.00),vTravel,z5,tPen\WObj:=wPaper;
    MoveL Offs(pOrigin,235.12,191.15,0.00),v60,z0,tPen\WObj:=wPaper;
    MoveL Offs(pOrigin,234.70,191.57,0.00),v40,z0,tPen\WObj:=wPaper;
    MoveL Offs(pOrigin,235.12,191.15,0.00),v40,fine,tPen\WObj:=wPaper;
    MoveL Offs(pOrigin,235.12,191.15,6.00),v60,z5,tPen\WObj:=wPaper;
    MoveL Offs(pOrigin,234.06,190.30,6.00),vTravel,z5,tPen\WObj:=wPaper;
    MoveL Offs(pOrigin,234.06,190.30,0.00),v60,z0,tPen\WObj:=wPaper;
    MoveL Offs(pOrigin,233.43,191.15,0.00),v40,z0,tPen\WObj:=wPaper;
    MoveL Offs(pOrigin,234.06,190.30,0.00),v40,fine,tPen\WObj:=wPaper;
    MoveL Offs(pOrigin,234.06,190.30,6.00),v60,z5,tPen\WObj:=wPaper;
    MoveL Offs(pOrigin,233.85,187.32,6.00),vTravel,z5,tPen\WObj:=wPaper;
    MoveL Offs(pOrigin,233.85,187.32,0.00),v60,z0,tPen\WObj:=wPaper;
    MoveL Offs(pOrigin,231.73,187.18,0.00),v40,z0,tPen\WObj:=wPaper;
    MoveL Offs(pOrigin,230.38,185.62,0.00),v40,z0,tPen\WObj:=wPaper;
    MoveL Offs(pOrigin,229.81,182.65,0.00),v40,z0,tPen\WObj:=wPaper;
    MoveL Offs(pOrigin,229.81,180.74,0.00),v40,z0,tPen\WObj:=wPaper;
    MoveL Offs(pOrigin,230.31,179.25,0.00),v40,z0,tPen\WObj:=wPaper;
    MoveL Offs(pOrigin,230.88,178.82,0.00),v40,z0,tPen\WObj:=wPaper;
    MoveL Offs(pOrigin,230.24,179.04,0.00),v40,z0,tPen\WObj:=wPaper;
    MoveL Offs(pOrigin,229.60,178.19,0.00),v40,z0,tPen\WObj:=wPaper;
    MoveL Offs(pOrigin,229.39,175.43,0.00),v40,z0,tPen\WObj:=wPaper;
    MoveL Offs(pOrigin,228.54,171.39,0.00),v40,z0,tPen\WObj:=wPaper;
    MoveL Offs(pOrigin,229.39,167.14,0.00),v40,z0,tPen\WObj:=wPaper;
    MoveL Offs(pOrigin,229.39,167.14,0.00),v40,z0,tPen\WObj:=wPaper;
    MoveL Offs(pOrigin,229.88,166.50,0.00),v40,z0,tPen\WObj:=wPaper;
    MoveL Offs(pOrigin,230.66,163.95,0.00),v40,z0,tPen\WObj:=wPaper;
    MoveL Offs(pOrigin,230.66,163.95,0.00),v40,z0,tPen\WObj:=wPaper;
    MoveL Offs(pOrigin,231.09,163.52,0.00),v40,z0,tPen\WObj:=wPaper;
    MoveL Offs(pOrigin,231.09,162.68,0.00),v40,z0,tPen\WObj:=wPaper;
    MoveL Offs(pOrigin,231.09,162.68,0.00),v40,z0,tPen\WObj:=wPaper;
    MoveL Offs(pOrigin,231.30,161.40,0.00),v40,z0,tPen\WObj:=wPaper;
    MoveL Offs(pOrigin,231.51,161.33,0.00),v40,z0,tPen\WObj:=wPaper;
    MoveL Offs(pOrigin,231.37,160.55,0.00),v40,z0,tPen\WObj:=wPaper;
    MoveL Offs(pOrigin,232.08,160.20,0.00),v40,z0,tPen\WObj:=wPaper;
    MoveL Offs(pOrigin,232.08,160.98,0.00),v40,z0,tPen\WObj:=wPaper;
    MoveL Offs(pOrigin,231.51,161.33,0.00),v40,fine,tPen\WObj:=wPaper;
    MoveL Offs(pOrigin,231.51,161.33,6.00),v60,z5,tPen\WObj:=wPaper;
    MoveL Offs(pOrigin,232.15,160.12,6.00),vTravel,z5,tPen\WObj:=wPaper;
    MoveL Offs(pOrigin,232.15,160.12,0.00),v60,z0,tPen\WObj:=wPaper;
    MoveL Offs(pOrigin,240.65,138.45,0.00),v40,z0,tPen\WObj:=wPaper;
    MoveL Offs(pOrigin,240.65,137.60,0.00),v40,fine,tPen\WObj:=wPaper;
    MoveL Offs(pOrigin,240.65,137.60,6.00),v60,z5,tPen\WObj:=wPaper;
    MoveL Offs(pOrigin,244.48,136.96,6.00),vTravel,z5,tPen\WObj:=wPaper;
    MoveL Offs(pOrigin,244.48,136.96,0.00),v60,z0,tPen\WObj:=wPaper;
    MoveL Offs(pOrigin,244.26,137.81,0.00),v40,z0,tPen\WObj:=wPaper;
    MoveL Offs(pOrigin,244.69,138.24,0.00),v40,fine,tPen\WObj:=wPaper;
    MoveL Offs(pOrigin,244.69,138.24,6.00),v60,z5,tPen\WObj:=wPaper;
    MoveL Offs(pOrigin,244.69,140.79,6.00),vTravel,z5,tPen\WObj:=wPaper;
    MoveL Offs(pOrigin,244.69,140.79,0.00),v60,z0,tPen\WObj:=wPaper;
    MoveL Offs(pOrigin,244.48,141.85,0.00),v40,z0,tPen\WObj:=wPaper;
    MoveL Offs(pOrigin,244.90,142.27,0.00),v40,z0,tPen\WObj:=wPaper;
    MoveL Offs(pOrigin,244.90,143.34,0.00),v40,z0,tPen\WObj:=wPaper;
    MoveL Offs(pOrigin,244.69,144.40,0.00),v40,z0,tPen\WObj:=wPaper;
    MoveL Offs(pOrigin,245.11,144.82,0.00),v40,z0,tPen\WObj:=wPaper;
    MoveL Offs(pOrigin,245.11,145.68,0.00),v40,z0,tPen\WObj:=wPaper;
    MoveL Offs(pOrigin,244.90,146.74,0.00),v40,z0,tPen\WObj:=wPaper;
    MoveL Offs(pOrigin,245.32,147.16,0.00),v40,z0,tPen\WObj:=wPaper;
    MoveL Offs(pOrigin,245.32,147.59,0.00),v40,z0,tPen\WObj:=wPaper;
    MoveL Offs(pOrigin,245.75,146.31,0.00),v40,z0,tPen\WObj:=wPaper;
    MoveL Offs(pOrigin,245.11,145.25,0.00),v40,z0,tPen\WObj:=wPaper;
    MoveL Offs(pOrigin,245.54,144.40,0.00),v40,z0,tPen\WObj:=wPaper;
    MoveL Offs(pOrigin,244.90,142.91,0.00),v40,z0,tPen\WObj:=wPaper;
    MoveL Offs(pOrigin,245.32,141.43,0.00),v40,z0,tPen\WObj:=wPaper;
    MoveL Offs(pOrigin,244.69,140.36,0.00),v40,z0,tPen\WObj:=wPaper;
    MoveL Offs(pOrigin,244.69,138.66,0.00),v40,z0,tPen\WObj:=wPaper;
    MoveL Offs(pOrigin,245.11,137.60,0.00),v40,z0,tPen\WObj:=wPaper;
    MoveL Offs(pOrigin,244.48,136.54,0.00),v40,z0,tPen\WObj:=wPaper;
    MoveL Offs(pOrigin,243.41,97.86,0.00),v40,z0,tPen\WObj:=wPaper;
    MoveL Offs(pOrigin,241.93,75.76,0.00),v40,z0,tPen\WObj:=wPaper;
    MoveL Offs(pOrigin,239.38,51.54,0.00),v40,z0,tPen\WObj:=wPaper;
    MoveL Offs(pOrigin,238.74,40.91,0.00),v40,z0,tPen\WObj:=wPaper;
    MoveL Offs(pOrigin,238.74,40.91,0.00),v40,z0,tPen\WObj:=wPaper;
    MoveL Offs(pOrigin,239.16,40.49,0.00),v40,z0,tPen\WObj:=wPaper;
    MoveL Offs(pOrigin,240.65,40.28,0.00),v40,z0,tPen\WObj:=wPaper;
    MoveL Offs(pOrigin,242.35,40.49,0.00),v40,z0,tPen\WObj:=wPaper;
    MoveL Offs(pOrigin,245.75,45.16,0.00),v40,z0,tPen\WObj:=wPaper;
    MoveL Offs(pOrigin,254.46,54.30,0.00),v40,z0,tPen\WObj:=wPaper;
    MoveL Offs(pOrigin,254.89,55.36,0.00),v40,z0,tPen\WObj:=wPaper;
    MoveL Offs(pOrigin,254.89,55.36,0.00),v40,z0,tPen\WObj:=wPaper;
    MoveL Offs(pOrigin,257.44,79.80,0.00),v40,z0,tPen\WObj:=wPaper;
    MoveL Offs(pOrigin,258.08,89.36,0.00),v40,z0,tPen\WObj:=wPaper;
    MoveL Offs(pOrigin,258.08,89.36,0.00),v40,z0,tPen\WObj:=wPaper;
  ENDPROC

  PROC DrawPart52()
    MoveL Offs(pOrigin,258.50,89.57,0.00),v40,z0,tPen\WObj:=wPaper;
    MoveL Offs(pOrigin,258.50,90.43,0.00),v40,z0,tPen\WObj:=wPaper;
    MoveL Offs(pOrigin,257.86,90.64,0.00),v40,z0,tPen\WObj:=wPaper;
    MoveL Offs(pOrigin,257.86,90.64,0.00),v40,z0,tPen\WObj:=wPaper;
    MoveL Offs(pOrigin,258.92,94.04,0.00),v40,z0,tPen\WObj:=wPaper;
    MoveL Offs(pOrigin,258.92,94.04,0.00),v40,z0,tPen\WObj:=wPaper;
    MoveL Offs(pOrigin,260.06,95.10,0.00),v40,z0,tPen\WObj:=wPaper;
    MoveL Offs(pOrigin,263.67,102.54,0.00),v40,z0,tPen\WObj:=wPaper;
    MoveL Offs(pOrigin,269.34,116.78,0.00),v40,fine,tPen\WObj:=wPaper;
    MoveL Offs(pOrigin,269.34,116.78,6.00),v60,z5,tPen\WObj:=wPaper;
    MoveL Offs(pOrigin,253.75,114.44,6.00),vTravel,z5,tPen\WObj:=wPaper;
    MoveL Offs(pOrigin,253.75,114.44,0.00),v60,z0,tPen\WObj:=wPaper;
    MoveL Offs(pOrigin,254.04,112.74,0.00),v40,z0,tPen\WObj:=wPaper;
    MoveL Offs(pOrigin,253.75,111.89,0.00),v40,z0,tPen\WObj:=wPaper;
    MoveL Offs(pOrigin,252.76,110.75,0.00),v40,z0,tPen\WObj:=wPaper;
    MoveL Offs(pOrigin,251.91,110.40,0.00),v40,z0,tPen\WObj:=wPaper;
    MoveL Offs(pOrigin,250.43,110.40,0.00),v40,z0,tPen\WObj:=wPaper;
    MoveL Offs(pOrigin,249.36,110.82,0.00),v40,z0,tPen\WObj:=wPaper;
    MoveL Offs(pOrigin,248.65,111.68,0.00),v40,z0,tPen\WObj:=wPaper;
    MoveL Offs(pOrigin,248.30,113.80,0.00),v40,z0,tPen\WObj:=wPaper;
    MoveL Offs(pOrigin,249.36,115.50,0.00),v40,z0,tPen\WObj:=wPaper;
    MoveL Offs(pOrigin,251.49,116.14,0.00),v40,z0,tPen\WObj:=wPaper;
    MoveL Offs(pOrigin,253.19,115.29,0.00),v40,z0,tPen\WObj:=wPaper;
    MoveL Offs(pOrigin,253.75,114.44,0.00),v40,z0,tPen\WObj:=wPaper;
    MoveL Offs(pOrigin,253.19,115.07,0.00),v40,z0,tPen\WObj:=wPaper;
    MoveL Offs(pOrigin,252.76,115.50,0.00),v40,z0,tPen\WObj:=wPaper;
    MoveL Offs(pOrigin,253.19,115.07,0.00),v40,fine,tPen\WObj:=wPaper;
    MoveL Offs(pOrigin,253.19,115.07,6.00),v60,z5,tPen\WObj:=wPaper;
    MoveL Offs(pOrigin,250.43,113.80,6.00),vTravel,z5,tPen\WObj:=wPaper;
    MoveL Offs(pOrigin,250.43,113.80,0.00),v60,z0,tPen\WObj:=wPaper;
    MoveL Offs(pOrigin,251.70,113.59,0.00),v40,z0,tPen\WObj:=wPaper;
    MoveL Offs(pOrigin,251.49,112.81,0.00),v40,z0,tPen\WObj:=wPaper;
    MoveL Offs(pOrigin,250.64,112.74,0.00),v40,fine,tPen\WObj:=wPaper;
    MoveL Offs(pOrigin,250.64,112.74,6.00),v60,z5,tPen\WObj:=wPaper;
    MoveL Offs(pOrigin,238.31,121.88,6.00),vTravel,z5,tPen\WObj:=wPaper;
    MoveL Offs(pOrigin,238.31,121.88,0.00),v60,z0,tPen\WObj:=wPaper;
    MoveL Offs(pOrigin,237.04,129.10,0.00),v40,z0,tPen\WObj:=wPaper;
    MoveL Offs(pOrigin,233.85,142.70,0.00),v40,fine,tPen\WObj:=wPaper;
    MoveL Offs(pOrigin,233.85,142.70,6.00),v60,z5,tPen\WObj:=wPaper;
    MoveL Offs(pOrigin,245.32,147.73,6.00),vTravel,z5,tPen\WObj:=wPaper;
    MoveL Offs(pOrigin,245.32,147.73,0.00),v60,z0,tPen\WObj:=wPaper;
    MoveL Offs(pOrigin,245.96,148.23,0.00),v40,z0,tPen\WObj:=wPaper;
    MoveL Offs(pOrigin,245.68,148.93,0.00),v40,z0,tPen\WObj:=wPaper;
    MoveL Offs(pOrigin,245.11,148.23,0.00),v40,z0,tPen\WObj:=wPaper;
    MoveL Offs(pOrigin,245.32,147.73,0.00),v40,fine,tPen\WObj:=wPaper;
    MoveL Offs(pOrigin,245.32,147.73,6.00),v60,z5,tPen\WObj:=wPaper;
    MoveL Offs(pOrigin,245.54,150.56,6.00),vTravel,z5,tPen\WObj:=wPaper;
    MoveL Offs(pOrigin,245.54,150.56,0.00),v60,z0,tPen\WObj:=wPaper;
    MoveL Offs(pOrigin,245.75,151.84,0.00),v40,z0,tPen\WObj:=wPaper;
    MoveL Offs(pOrigin,246.39,151.84,0.00),v40,z0,tPen\WObj:=wPaper;
    MoveL Offs(pOrigin,246.18,150.56,0.00),v40,z0,tPen\WObj:=wPaper;
    MoveL Offs(pOrigin,246.18,150.56,0.00),v40,z0,tPen\WObj:=wPaper;
    MoveL Offs(pOrigin,246.10,149.50,0.00),v40,z0,tPen\WObj:=wPaper;
    MoveL Offs(pOrigin,245.54,149.22,0.00),v40,z0,tPen\WObj:=wPaper;
    MoveL Offs(pOrigin,245.32,149.93,0.00),v40,z0,tPen\WObj:=wPaper;
    MoveL Offs(pOrigin,245.54,150.56,0.00),v40,fine,tPen\WObj:=wPaper;
    MoveL Offs(pOrigin,245.54,150.56,6.00),v60,z5,tPen\WObj:=wPaper;
    MoveL Offs(pOrigin,250.64,152.05,6.00),vTravel,z5,tPen\WObj:=wPaper;
    MoveL Offs(pOrigin,250.64,152.05,0.00),v60,z0,tPen\WObj:=wPaper;
    MoveL Offs(pOrigin,250.64,153.54,0.00),v40,z0,tPen\WObj:=wPaper;
    MoveL Offs(pOrigin,251.27,154.81,0.00),v40,z0,tPen\WObj:=wPaper;
    MoveL Offs(pOrigin,251.91,155.31,0.00),v40,z0,tPen\WObj:=wPaper;
    MoveL Offs(pOrigin,254.04,155.66,0.00),v40,z0,tPen\WObj:=wPaper;
    MoveL Offs(pOrigin,255.60,154.60,0.00),v40,z0,tPen\WObj:=wPaper;
    MoveL Offs(pOrigin,256.16,153.32,0.00),v40,z0,tPen\WObj:=wPaper;
    MoveL Offs(pOrigin,256.16,152.48,0.00),v40,z0,tPen\WObj:=wPaper;
    MoveL Offs(pOrigin,255.81,151.41,0.00),v40,z0,tPen\WObj:=wPaper;
    MoveL Offs(pOrigin,254.89,150.35,0.00),v40,z0,tPen\WObj:=wPaper;
    MoveL Offs(pOrigin,252.98,149.93,0.00),v40,z0,tPen\WObj:=wPaper;
    MoveL Offs(pOrigin,251.20,150.99,0.00),v40,z0,tPen\WObj:=wPaper;
    MoveL Offs(pOrigin,250.64,152.05,0.00),v40,fine,tPen\WObj:=wPaper;
    MoveL Offs(pOrigin,250.64,152.05,6.00),v60,z5,tPen\WObj:=wPaper;
    MoveL Offs(pOrigin,252.98,152.26,6.00),vTravel,z5,tPen\WObj:=wPaper;
    MoveL Offs(pOrigin,252.98,152.26,0.00),v60,z0,tPen\WObj:=wPaper;
    MoveL Offs(pOrigin,253.82,152.48,0.00),v40,z0,tPen\WObj:=wPaper;
    MoveL Offs(pOrigin,254.04,153.11,0.00),v40,z0,tPen\WObj:=wPaper;
    MoveL Offs(pOrigin,253.61,153.54,0.00),v40,z0,tPen\WObj:=wPaper;
    MoveL Offs(pOrigin,252.76,153.54,0.00),v40,fine,tPen\WObj:=wPaper;
    MoveL Offs(pOrigin,252.76,153.54,6.00),v60,z5,tPen\WObj:=wPaper;
    MoveL Offs(pOrigin,249.15,158.00,6.00),vTravel,z5,tPen\WObj:=wPaper;
    MoveL Offs(pOrigin,249.15,158.00,0.00),v60,z0,tPen\WObj:=wPaper;
    MoveL Offs(pOrigin,249.79,158.85,0.00),v40,z0,tPen\WObj:=wPaper;
    MoveL Offs(pOrigin,249.15,158.00,0.00),v40,fine,tPen\WObj:=wPaper;
    MoveL Offs(pOrigin,249.15,158.00,6.00),v60,z5,tPen\WObj:=wPaper;
    MoveL Offs(pOrigin,249.57,160.55,6.00),vTravel,z5,tPen\WObj:=wPaper;
    MoveL Offs(pOrigin,249.57,160.55,0.00),v60,z0,tPen\WObj:=wPaper;
    MoveL Offs(pOrigin,250.00,160.98,0.00),v40,z0,tPen\WObj:=wPaper;
    MoveL Offs(pOrigin,249.57,160.55,0.00),v40,fine,tPen\WObj:=wPaper;
    MoveL Offs(pOrigin,249.57,160.55,6.00),v60,z5,tPen\WObj:=wPaper;
    MoveL Offs(pOrigin,250.85,162.04,6.00),vTravel,z5,tPen\WObj:=wPaper;
    MoveL Offs(pOrigin,250.85,162.04,0.00),v60,z0,tPen\WObj:=wPaper;
    MoveL Offs(pOrigin,251.70,162.89,0.00),v40,z0,tPen\WObj:=wPaper;
    MoveL Offs(pOrigin,250.85,162.04,0.00),v40,fine,tPen\WObj:=wPaper;
    MoveL Offs(pOrigin,250.85,162.04,6.00),v60,z5,tPen\WObj:=wPaper;
    MoveL Offs(pOrigin,251.27,164.38,6.00),vTravel,z5,tPen\WObj:=wPaper;
    MoveL Offs(pOrigin,251.27,164.38,0.00),v60,z0,tPen\WObj:=wPaper;
    MoveL Offs(pOrigin,250.64,165.01,0.00),v40,z0,tPen\WObj:=wPaper;
    MoveL Offs(pOrigin,251.27,164.38,0.00),v40,fine,tPen\WObj:=wPaper;
    MoveL Offs(pOrigin,251.27,164.38,6.00),v60,z5,tPen\WObj:=wPaper;
    MoveL Offs(pOrigin,252.34,165.01,6.00),vTravel,z5,tPen\WObj:=wPaper;
    MoveL Offs(pOrigin,252.34,165.01,0.00),v60,z0,tPen\WObj:=wPaper;
    MoveL Offs(pOrigin,252.12,165.44,0.00),v40,z0,tPen\WObj:=wPaper;
    MoveL Offs(pOrigin,252.34,165.01,0.00),v40,fine,tPen\WObj:=wPaper;
    MoveL Offs(pOrigin,252.34,165.01,6.00),v60,z5,tPen\WObj:=wPaper;
    MoveL Offs(pOrigin,253.61,164.80,6.00),vTravel,z5,tPen\WObj:=wPaper;
    MoveL Offs(pOrigin,253.61,164.80,0.00),v60,z0,tPen\WObj:=wPaper;
    MoveL Offs(pOrigin,254.04,165.23,0.00),v40,z0,tPen\WObj:=wPaper;
    MoveL Offs(pOrigin,253.61,164.80,0.00),v40,z0,tPen\WObj:=wPaper;
    MoveL Offs(pOrigin,254.25,165.44,0.00),v40,z0,tPen\WObj:=wPaper;
    MoveL Offs(pOrigin,254.68,165.86,0.00),v40,z0,tPen\WObj:=wPaper;
    MoveL Offs(pOrigin,254.25,165.44,0.00),v40,fine,tPen\WObj:=wPaper;
    MoveL Offs(pOrigin,254.25,165.44,6.00),v60,z5,tPen\WObj:=wPaper;
    MoveL Offs(pOrigin,255.74,166.71,6.00),vTravel,z5,tPen\WObj:=wPaper;
    MoveL Offs(pOrigin,255.74,166.71,0.00),v60,z0,tPen\WObj:=wPaper;
    MoveL Offs(pOrigin,257.86,168.84,0.00),v40,z0,tPen\WObj:=wPaper;
    MoveL Offs(pOrigin,255.74,166.71,0.00),v40,fine,tPen\WObj:=wPaper;
    MoveL Offs(pOrigin,255.74,166.71,6.00),v60,z5,tPen\WObj:=wPaper;
    MoveL Offs(pOrigin,256.59,165.65,6.00),vTravel,z5,tPen\WObj:=wPaper;
    MoveL Offs(pOrigin,256.59,165.65,0.00),v60,z0,tPen\WObj:=wPaper;
    MoveL Offs(pOrigin,257.01,166.07,0.00),v40,z0,tPen\WObj:=wPaper;
  ENDPROC

  PROC DrawPart53()
    MoveL Offs(pOrigin,256.59,165.65,0.00),v40,fine,tPen\WObj:=wPaper;
    MoveL Offs(pOrigin,256.59,165.65,6.00),v60,z5,tPen\WObj:=wPaper;
    MoveL Offs(pOrigin,258.92,167.99,6.00),vTravel,z5,tPen\WObj:=wPaper;
    MoveL Offs(pOrigin,258.92,167.99,0.00),v60,z0,tPen\WObj:=wPaper;
    MoveL Offs(pOrigin,259.35,168.41,0.00),v40,z0,tPen\WObj:=wPaper;
    MoveL Offs(pOrigin,258.92,167.99,0.00),v40,fine,tPen\WObj:=wPaper;
    MoveL Offs(pOrigin,258.92,167.99,6.00),v60,z5,tPen\WObj:=wPaper;
    MoveL Offs(pOrigin,258.71,170.11,6.00),vTravel,z5,tPen\WObj:=wPaper;
    MoveL Offs(pOrigin,258.71,170.11,0.00),v60,z0,tPen\WObj:=wPaper;
    MoveL Offs(pOrigin,258.92,170.54,0.00),v40,z0,tPen\WObj:=wPaper;
    MoveL Offs(pOrigin,258.71,170.11,0.00),v40,fine,tPen\WObj:=wPaper;
    MoveL Offs(pOrigin,258.71,170.11,6.00),v60,z5,tPen\WObj:=wPaper;
    MoveL Offs(pOrigin,262.33,166.07,6.00),vTravel,z5,tPen\WObj:=wPaper;
    MoveL Offs(pOrigin,262.33,166.07,0.00),v60,z0,tPen\WObj:=wPaper;
    MoveL Offs(pOrigin,261.05,159.06,0.00),v40,z0,tPen\WObj:=wPaper;
    MoveL Offs(pOrigin,260.41,150.56,0.00),v40,z0,tPen\WObj:=wPaper;
    MoveL Offs(pOrigin,259.35,110.82,0.00),v40,z0,tPen\WObj:=wPaper;
    MoveL Offs(pOrigin,258.50,94.46,0.00),v40,z0,tPen\WObj:=wPaper;
    MoveL Offs(pOrigin,258.92,94.04,0.00),v40,fine,tPen\WObj:=wPaper;
    MoveL Offs(pOrigin,258.92,94.04,6.00),v60,z5,tPen\WObj:=wPaper;
    MoveL Offs(pOrigin,260.20,95.10,6.00),vTravel,z5,tPen\WObj:=wPaper;
    MoveL Offs(pOrigin,260.20,95.10,0.00),v60,z0,tPen\WObj:=wPaper;
    MoveL Offs(pOrigin,260.41,95.53,0.00),v40,z0,tPen\WObj:=wPaper;
    MoveL Offs(pOrigin,260.20,95.10,0.00),v40,fine,tPen\WObj:=wPaper;
    MoveL Offs(pOrigin,260.20,95.10,6.00),v60,z5,tPen\WObj:=wPaper;
    MoveL Offs(pOrigin,261.05,96.80,6.00),vTravel,z5,tPen\WObj:=wPaper;
    MoveL Offs(pOrigin,261.05,96.80,0.00),v60,z0,tPen\WObj:=wPaper;
    MoveL Offs(pOrigin,261.26,97.22,0.00),v40,z0,tPen\WObj:=wPaper;
    MoveL Offs(pOrigin,261.05,96.80,0.00),v40,z0,tPen\WObj:=wPaper;
    MoveL Offs(pOrigin,261.48,97.65,0.00),v40,z0,tPen\WObj:=wPaper;
    MoveL Offs(pOrigin,261.69,98.07,0.00),v40,z0,tPen\WObj:=wPaper;
    MoveL Offs(pOrigin,261.48,97.65,0.00),v40,fine,tPen\WObj:=wPaper;
    MoveL Offs(pOrigin,261.48,97.65,6.00),v60,z5,tPen\WObj:=wPaper;
    MoveL Offs(pOrigin,262.11,99.14,6.00),vTravel,z5,tPen\WObj:=wPaper;
    MoveL Offs(pOrigin,262.11,99.14,0.00),v60,z0,tPen\WObj:=wPaper;
    MoveL Offs(pOrigin,262.33,99.56,0.00),v40,z0,tPen\WObj:=wPaper;
    MoveL Offs(pOrigin,262.11,99.14,0.00),v40,fine,tPen\WObj:=wPaper;
    MoveL Offs(pOrigin,262.11,99.14,6.00),v60,z5,tPen\WObj:=wPaper;
    MoveL Offs(pOrigin,257.86,90.64,6.00),vTravel,z5,tPen\WObj:=wPaper;
    MoveL Offs(pOrigin,257.86,90.64,0.00),v60,z0,tPen\WObj:=wPaper;
    MoveL Offs(pOrigin,257.44,90.43,0.00),v40,z0,tPen\WObj:=wPaper;
    MoveL Offs(pOrigin,257.23,89.57,0.00),v40,z0,tPen\WObj:=wPaper;
    MoveL Offs(pOrigin,257.23,89.57,0.00),v40,z0,tPen\WObj:=wPaper;
    MoveL Offs(pOrigin,252.12,81.50,0.00),v40,fine,tPen\WObj:=wPaper;
    MoveL Offs(pOrigin,252.12,81.50,6.00),v60,z5,tPen\WObj:=wPaper;
    MoveL Offs(pOrigin,249.36,71.09,6.00),vTravel,z5,tPen\WObj:=wPaper;
    MoveL Offs(pOrigin,249.36,71.09,0.00),v60,z0,tPen\WObj:=wPaper;
    MoveL Offs(pOrigin,250.43,70.45,0.00),v40,z0,tPen\WObj:=wPaper;
    MoveL Offs(pOrigin,251.27,68.96,0.00),v40,z0,tPen\WObj:=wPaper;
    MoveL Offs(pOrigin,251.27,67.69,0.00),v40,z0,tPen\WObj:=wPaper;
    MoveL Offs(pOrigin,250.85,66.84,0.00),v40,z0,tPen\WObj:=wPaper;
    MoveL Offs(pOrigin,249.79,65.85,0.00),v40,z0,tPen\WObj:=wPaper;
    MoveL Offs(pOrigin,248.09,65.56,0.00),v40,z0,tPen\WObj:=wPaper;
    MoveL Offs(pOrigin,246.60,66.20,0.00),v40,z0,tPen\WObj:=wPaper;
    MoveL Offs(pOrigin,245.61,68.11,0.00),v40,z0,tPen\WObj:=wPaper;
    MoveL Offs(pOrigin,246.18,70.03,0.00),v40,z0,tPen\WObj:=wPaper;
    MoveL Offs(pOrigin,247.66,71.09,0.00),v40,z0,tPen\WObj:=wPaper;
    MoveL Offs(pOrigin,249.36,71.09,0.00),v40,fine,tPen\WObj:=wPaper;
    MoveL Offs(pOrigin,249.36,71.09,6.00),v60,z5,tPen\WObj:=wPaper;
    MoveL Offs(pOrigin,249.15,68.11,6.00),vTravel,z5,tPen\WObj:=wPaper;
    MoveL Offs(pOrigin,249.15,68.11,0.00),v60,z0,tPen\WObj:=wPaper;
    MoveL Offs(pOrigin,249.08,68.89,0.00),v40,z0,tPen\WObj:=wPaper;
    MoveL Offs(pOrigin,248.30,68.96,0.00),v40,z0,tPen\WObj:=wPaper;
    MoveL Offs(pOrigin,247.95,68.75,0.00),v40,z0,tPen\WObj:=wPaper;
    MoveL Offs(pOrigin,247.88,67.90,0.00),v40,fine,tPen\WObj:=wPaper;
    MoveL Offs(pOrigin,247.88,67.90,6.00),v60,z5,tPen\WObj:=wPaper;
    MoveL Offs(pOrigin,238.31,71.09,6.00),vTravel,z5,tPen\WObj:=wPaper;
    MoveL Offs(pOrigin,238.31,71.09,0.00),v60,z0,tPen\WObj:=wPaper;
    MoveL Offs(pOrigin,234.27,76.40,0.00),v40,z0,tPen\WObj:=wPaper;
    MoveL Offs(pOrigin,230.88,82.14,0.00),v40,z0,tPen\WObj:=wPaper;
    MoveL Offs(pOrigin,230.88,82.14,0.00),v40,z0,tPen\WObj:=wPaper;
    MoveL Offs(pOrigin,230.88,85.54,0.00),v40,z0,tPen\WObj:=wPaper;
    MoveL Offs(pOrigin,231.73,91.28,0.00),v40,z0,tPen\WObj:=wPaper;
    MoveL Offs(pOrigin,232.79,103.81,0.00),v40,z0,tPen\WObj:=wPaper;
    MoveL Offs(pOrigin,233.00,118.26,0.00),v40,z0,tPen\WObj:=wPaper;
    MoveL Offs(pOrigin,231.94,136.96,0.00),v40,z0,tPen\WObj:=wPaper;
    MoveL Offs(pOrigin,228.96,164.80,0.00),v40,fine,tPen\WObj:=wPaper;
    MoveL Offs(pOrigin,228.96,164.80,6.00),v60,z5,tPen\WObj:=wPaper;
    MoveL Offs(pOrigin,230.24,163.95,6.00),vTravel,z5,tPen\WObj:=wPaper;
    MoveL Offs(pOrigin,230.24,163.95,0.00),v60,z0,tPen\WObj:=wPaper;
    MoveL Offs(pOrigin,228.96,165.23,0.00),v40,z0,tPen\WObj:=wPaper;
    MoveL Offs(pOrigin,228.75,166.71,0.00),v40,z0,tPen\WObj:=wPaper;
    MoveL Offs(pOrigin,229.39,167.14,0.00),v40,fine,tPen\WObj:=wPaper;
    MoveL Offs(pOrigin,229.39,167.14,6.00),v60,z5,tPen\WObj:=wPaper;
    MoveL Offs(pOrigin,230.24,163.95,6.00),vTravel,z5,tPen\WObj:=wPaper;
    MoveL Offs(pOrigin,230.24,163.95,0.00),v60,z0,tPen\WObj:=wPaper;
    MoveL Offs(pOrigin,230.24,163.10,0.00),v40,z0,tPen\WObj:=wPaper;
    MoveL Offs(pOrigin,231.09,162.68,0.00),v40,fine,tPen\WObj:=wPaper;
    MoveL Offs(pOrigin,231.09,162.68,6.00),v60,z5,tPen\WObj:=wPaper;
    MoveL Offs(pOrigin,233.64,156.09,6.00),vTravel,z5,tPen\WObj:=wPaper;
    MoveL Offs(pOrigin,233.64,156.09,0.00),v60,z0,tPen\WObj:=wPaper;
    MoveL Offs(pOrigin,233.43,156.51,0.00),v40,z0,tPen\WObj:=wPaper;
    MoveL Offs(pOrigin,233.64,156.09,0.00),v40,fine,tPen\WObj:=wPaper;
    MoveL Offs(pOrigin,233.64,156.09,6.00),v60,z5,tPen\WObj:=wPaper;
    MoveL Offs(pOrigin,246.18,157.79,6.00),vTravel,z5,tPen\WObj:=wPaper;
    MoveL Offs(pOrigin,246.18,157.79,0.00),v60,z0,tPen\WObj:=wPaper;
    MoveL Offs(pOrigin,244.12,161.61,0.00),v40,z0,tPen\WObj:=wPaper;
    MoveL Offs(pOrigin,241.22,165.86,0.00),v40,z0,tPen\WObj:=wPaper;
    MoveL Offs(pOrigin,240.86,167.35,0.00),v40,z0,tPen\WObj:=wPaper;
    MoveL Offs(pOrigin,240.86,167.35,0.00),v40,z0,tPen\WObj:=wPaper;
    MoveL Offs(pOrigin,235.90,172.80,0.00),v40,z0,tPen\WObj:=wPaper;
    MoveL Offs(pOrigin,234.91,173.30,0.00),v40,z0,tPen\WObj:=wPaper;
    MoveL Offs(pOrigin,231.16,177.55,0.00),v40,z0,tPen\WObj:=wPaper;
    MoveL Offs(pOrigin,230.95,178.61,0.00),v40,z0,tPen\WObj:=wPaper;
    MoveL Offs(pOrigin,231.30,178.82,0.00),v40,z0,tPen\WObj:=wPaper;
    MoveL Offs(pOrigin,232.15,178.54,0.00),v40,z0,tPen\WObj:=wPaper;
    MoveL Offs(pOrigin,237.25,175.21,0.00),v40,fine,tPen\WObj:=wPaper;
    MoveL Offs(pOrigin,237.25,175.21,6.00),v60,z5,tPen\WObj:=wPaper;
    MoveL Offs(pOrigin,234.06,174.15,6.00),vTravel,z5,tPen\WObj:=wPaper;
    MoveL Offs(pOrigin,234.06,174.15,0.00),v60,z0,tPen\WObj:=wPaper;
    MoveL Offs(pOrigin,233.64,174.57,0.00),v40,z0,tPen\WObj:=wPaper;
    MoveL Offs(pOrigin,234.06,174.15,0.00),v40,fine,tPen\WObj:=wPaper;
    MoveL Offs(pOrigin,234.06,174.15,6.00),v60,z5,tPen\WObj:=wPaper;
    MoveL Offs(pOrigin,240.86,167.35,6.00),vTravel,z5,tPen\WObj:=wPaper;
    MoveL Offs(pOrigin,240.86,167.35,0.00),v60,z0,tPen\WObj:=wPaper;
    MoveL Offs(pOrigin,242.14,167.07,0.00),v40,z0,tPen\WObj:=wPaper;
    MoveL Offs(pOrigin,248.51,163.10,0.00),v40,fine,tPen\WObj:=wPaper;
    MoveL Offs(pOrigin,248.51,163.10,6.00),v60,z5,tPen\WObj:=wPaper;
    MoveL Offs(pOrigin,253.82,163.10,6.00),vTravel,z5,tPen\WObj:=wPaper;
    MoveL Offs(pOrigin,253.82,163.10,0.00),v60,z0,tPen\WObj:=wPaper;
  ENDPROC

  PROC DrawPart54()
    MoveL Offs(pOrigin,254.25,163.52,0.00),v40,z0,tPen\WObj:=wPaper;
    MoveL Offs(pOrigin,253.82,163.10,0.00),v40,fine,tPen\WObj:=wPaper;
    MoveL Offs(pOrigin,253.82,163.10,6.00),v60,z5,tPen\WObj:=wPaper;
    MoveL Offs(pOrigin,252.98,159.70,6.00),vTravel,z5,tPen\WObj:=wPaper;
    MoveL Offs(pOrigin,252.98,159.70,0.00),v60,z0,tPen\WObj:=wPaper;
    MoveL Offs(pOrigin,261.05,165.65,0.00),v40,z0,tPen\WObj:=wPaper;
    MoveL Offs(pOrigin,262.33,166.07,0.00),v40,z0,tPen\WObj:=wPaper;
    MoveL Offs(pOrigin,262.33,166.07,0.00),v40,z0,tPen\WObj:=wPaper;
    MoveL Offs(pOrigin,262.75,167.14,0.00),v40,z0,tPen\WObj:=wPaper;
    MoveL Offs(pOrigin,267.21,172.24,0.00),v40,z0,tPen\WObj:=wPaper;
    MoveL Offs(pOrigin,269.05,175.00,0.00),v40,z0,tPen\WObj:=wPaper;
    MoveL Offs(pOrigin,269.76,176.70,0.00),v40,z0,tPen\WObj:=wPaper;
    MoveL Offs(pOrigin,277.20,181.16,0.00),v40,fine,tPen\WObj:=wPaper;
    MoveL Offs(pOrigin,277.20,181.16,6.00),v60,z5,tPen\WObj:=wPaper;
    MoveL Offs(pOrigin,277.41,178.40,6.00),vTravel,z5,tPen\WObj:=wPaper;
    MoveL Offs(pOrigin,277.41,178.40,0.00),v60,z0,tPen\WObj:=wPaper;
    MoveL Offs(pOrigin,276.49,176.91,0.00),v40,z0,tPen\WObj:=wPaper;
    MoveL Offs(pOrigin,275.15,176.06,0.00),v40,z0,tPen\WObj:=wPaper;
    MoveL Offs(pOrigin,271.25,170.54,0.00),v40,fine,tPen\WObj:=wPaper;
    MoveL Offs(pOrigin,271.25,170.54,6.00),v60,z5,tPen\WObj:=wPaper;
    MoveL Offs(pOrigin,269.34,176.27,6.00),vTravel,z5,tPen\WObj:=wPaper;
    MoveL Offs(pOrigin,269.34,176.27,0.00),v60,z0,tPen\WObj:=wPaper;
    MoveL Offs(pOrigin,267.00,175.71,0.00),v40,z0,tPen\WObj:=wPaper;
    MoveL Offs(pOrigin,264.45,174.57,0.00),v40,z0,tPen\WObj:=wPaper;
    MoveL Offs(pOrigin,263.60,174.57,0.00),v40,fine,tPen\WObj:=wPaper;
    MoveL Offs(pOrigin,263.60,174.57,6.00),v60,z5,tPen\WObj:=wPaper;
    MoveL Offs(pOrigin,262.33,176.27,6.00),vTravel,z5,tPen\WObj:=wPaper;
    MoveL Offs(pOrigin,262.33,176.27,0.00),v60,z0,tPen\WObj:=wPaper;
    MoveL Offs(pOrigin,262.75,176.91,0.00),v40,z0,tPen\WObj:=wPaper;
    MoveL Offs(pOrigin,262.33,176.27,0.00),v40,fine,tPen\WObj:=wPaper;
    MoveL Offs(pOrigin,262.33,176.27,6.00),v60,z5,tPen\WObj:=wPaper;
    MoveL Offs(pOrigin,263.60,178.19,6.00),vTravel,z5,tPen\WObj:=wPaper;
    MoveL Offs(pOrigin,263.60,178.19,0.00),v60,z0,tPen\WObj:=wPaper;
    MoveL Offs(pOrigin,263.81,178.61,0.00),v40,z0,tPen\WObj:=wPaper;
    MoveL Offs(pOrigin,263.60,178.19,0.00),v40,fine,tPen\WObj:=wPaper;
    MoveL Offs(pOrigin,263.60,178.19,6.00),v60,z5,tPen\WObj:=wPaper;
    MoveL Offs(pOrigin,262.96,179.89,6.00),vTravel,z5,tPen\WObj:=wPaper;
    MoveL Offs(pOrigin,262.96,179.89,0.00),v60,z0,tPen\WObj:=wPaper;
    MoveL Offs(pOrigin,263.39,180.31,0.00),v40,z0,tPen\WObj:=wPaper;
    MoveL Offs(pOrigin,262.96,179.89,0.00),v40,fine,tPen\WObj:=wPaper;
    MoveL Offs(pOrigin,262.96,179.89,6.00),v60,z5,tPen\WObj:=wPaper;
    MoveL Offs(pOrigin,264.66,179.89,6.00),vTravel,z5,tPen\WObj:=wPaper;
    MoveL Offs(pOrigin,264.66,179.89,0.00),v60,z0,tPen\WObj:=wPaper;
    MoveL Offs(pOrigin,265.09,180.31,0.00),v40,z0,tPen\WObj:=wPaper;
    MoveL Offs(pOrigin,264.66,179.89,0.00),v40,fine,tPen\WObj:=wPaper;
    MoveL Offs(pOrigin,264.66,179.89,6.00),v60,z5,tPen\WObj:=wPaper;
    MoveL Offs(pOrigin,265.73,181.16,6.00),vTravel,z5,tPen\WObj:=wPaper;
    MoveL Offs(pOrigin,265.73,181.16,0.00),v60,z0,tPen\WObj:=wPaper;
    MoveL Offs(pOrigin,265.94,181.59,0.00),v40,z0,tPen\WObj:=wPaper;
    MoveL Offs(pOrigin,265.73,181.16,0.00),v40,fine,tPen\WObj:=wPaper;
    MoveL Offs(pOrigin,265.73,181.16,6.00),v60,z5,tPen\WObj:=wPaper;
    MoveL Offs(pOrigin,265.73,177.12,6.00),vTravel,z5,tPen\WObj:=wPaper;
    MoveL Offs(pOrigin,265.73,177.12,0.00),v60,z0,tPen\WObj:=wPaper;
    MoveL Offs(pOrigin,271.75,186.69,0.00),v40,z0,tPen\WObj:=wPaper;
    MoveL Offs(pOrigin,272.95,187.96,0.00),v40,z0,tPen\WObj:=wPaper;
    MoveL Offs(pOrigin,272.95,187.96,0.00),v40,z0,tPen\WObj:=wPaper;
    MoveL Offs(pOrigin,273.02,188.60,0.00),v40,z0,tPen\WObj:=wPaper;
    MoveL Offs(pOrigin,274.01,189.02,0.00),v40,z0,tPen\WObj:=wPaper;
    MoveL Offs(pOrigin,275.29,188.88,0.00),v40,z0,tPen\WObj:=wPaper;
    MoveL Offs(pOrigin,276.77,187.96,0.00),v40,z0,tPen\WObj:=wPaper;
    MoveL Offs(pOrigin,278.05,184.99,0.00),v40,z0,tPen\WObj:=wPaper;
    MoveL Offs(pOrigin,279.82,177.34,0.00),v40,z0,tPen\WObj:=wPaper;
    MoveL Offs(pOrigin,280.39,177.20,0.00),v40,z0,tPen\WObj:=wPaper;
    MoveL Offs(pOrigin,287.61,206.45,0.00),v40,z0,tPen\WObj:=wPaper;
    MoveL Offs(pOrigin,288.67,215.38,0.00),v40,z0,tPen\WObj:=wPaper;
    MoveL Offs(pOrigin,288.67,219.41,0.00),v40,z0,tPen\WObj:=wPaper;
    MoveL Offs(pOrigin,288.25,220.90,0.00),v40,fine,tPen\WObj:=wPaper;
    MoveL Offs(pOrigin,288.25,220.90,6.00),v60,z5,tPen\WObj:=wPaper;
    MoveL Offs(pOrigin,286.55,222.39,6.00),vTravel,z5,tPen\WObj:=wPaper;
    MoveL Offs(pOrigin,286.55,222.39,0.00),v60,z0,tPen\WObj:=wPaper;
    MoveL Offs(pOrigin,285.91,221.96,0.00),v40,z0,tPen\WObj:=wPaper;
    MoveL Offs(pOrigin,284.42,219.84,0.00),v40,z0,tPen\WObj:=wPaper;
    MoveL Offs(pOrigin,283.79,219.48,0.00),v40,z0,tPen\WObj:=wPaper;
    MoveL Offs(pOrigin,283.43,219.62,0.00),v40,z0,tPen\WObj:=wPaper;
    MoveL Offs(pOrigin,285.91,223.45,0.00),v40,z0,tPen\WObj:=wPaper;
    MoveL Offs(pOrigin,286.55,223.88,0.00),v40,fine,tPen\WObj:=wPaper;
    MoveL Offs(pOrigin,286.55,223.88,6.00),v60,z5,tPen\WObj:=wPaper;
    MoveL Offs(pOrigin,287.40,226.00,6.00),vTravel,z5,tPen\WObj:=wPaper;
    MoveL Offs(pOrigin,287.40,226.00,0.00),v60,z0,tPen\WObj:=wPaper;
    MoveL Offs(pOrigin,287.61,226.43,0.00),v40,z0,tPen\WObj:=wPaper;
    MoveL Offs(pOrigin,287.40,226.00,0.00),v40,z0,tPen\WObj:=wPaper;
    MoveL Offs(pOrigin,287.83,226.85,0.00),v40,z0,tPen\WObj:=wPaper;
    MoveL Offs(pOrigin,288.04,227.27,0.00),v40,z0,tPen\WObj:=wPaper;
    MoveL Offs(pOrigin,287.83,226.85,0.00),v40,fine,tPen\WObj:=wPaper;
    MoveL Offs(pOrigin,287.83,226.85,6.00),v60,z5,tPen\WObj:=wPaper;
    MoveL Offs(pOrigin,292.08,222.81,6.00),vTravel,z5,tPen\WObj:=wPaper;
    MoveL Offs(pOrigin,292.08,222.81,0.00),v60,z0,tPen\WObj:=wPaper;
    MoveL Offs(pOrigin,291.86,223.24,0.00),v40,z0,tPen\WObj:=wPaper;
    MoveL Offs(pOrigin,292.08,222.81,0.00),v40,z0,tPen\WObj:=wPaper;
    MoveL Offs(pOrigin,292.71,222.18,0.00),v40,z0,tPen\WObj:=wPaper;
    MoveL Offs(pOrigin,292.50,222.60,0.00),v40,z0,tPen\WObj:=wPaper;
    MoveL Offs(pOrigin,292.71,222.18,0.00),v40,fine,tPen\WObj:=wPaper;
    MoveL Offs(pOrigin,292.71,222.18,6.00),v60,z5,tPen\WObj:=wPaper;
    MoveL Offs(pOrigin,291.65,221.32,6.00),vTravel,z5,tPen\WObj:=wPaper;
    MoveL Offs(pOrigin,291.65,221.32,0.00),v60,z0,tPen\WObj:=wPaper;
    MoveL Offs(pOrigin,291.01,221.96,0.00),v40,z0,tPen\WObj:=wPaper;
    MoveL Offs(pOrigin,291.65,221.32,0.00),v40,fine,tPen\WObj:=wPaper;
    MoveL Offs(pOrigin,291.65,221.32,6.00),v60,z5,tPen\WObj:=wPaper;
    MoveL Offs(pOrigin,292.50,220.26,6.00),vTravel,z5,tPen\WObj:=wPaper;
    MoveL Offs(pOrigin,292.50,220.26,0.00),v60,z0,tPen\WObj:=wPaper;
    MoveL Offs(pOrigin,292.08,220.69,0.00),v40,z0,tPen\WObj:=wPaper;
    MoveL Offs(pOrigin,292.50,220.26,0.00),v40,fine,tPen\WObj:=wPaper;
    MoveL Offs(pOrigin,292.50,220.26,6.00),v60,z5,tPen\WObj:=wPaper;
    MoveL Offs(pOrigin,293.56,221.11,6.00),vTravel,z5,tPen\WObj:=wPaper;
    MoveL Offs(pOrigin,293.56,221.11,0.00),v60,z0,tPen\WObj:=wPaper;
    MoveL Offs(pOrigin,293.35,221.54,0.00),v40,z0,tPen\WObj:=wPaper;
    MoveL Offs(pOrigin,293.56,221.11,0.00),v40,fine,tPen\WObj:=wPaper;
    MoveL Offs(pOrigin,293.56,221.11,6.00),v60,z5,tPen\WObj:=wPaper;
    MoveL Offs(pOrigin,294.41,220.26,6.00),vTravel,z5,tPen\WObj:=wPaper;
    MoveL Offs(pOrigin,294.41,220.26,0.00),v60,z0,tPen\WObj:=wPaper;
    MoveL Offs(pOrigin,294.62,219.84,0.00),v40,z0,tPen\WObj:=wPaper;
    MoveL Offs(pOrigin,294.41,220.26,0.00),v40,z0,tPen\WObj:=wPaper;
    MoveL Offs(pOrigin,295.05,219.62,0.00),v40,z0,tPen\WObj:=wPaper;
    MoveL Offs(pOrigin,295.26,219.20,0.00),v40,z0,tPen\WObj:=wPaper;
    MoveL Offs(pOrigin,295.05,219.62,0.00),v40,fine,tPen\WObj:=wPaper;
    MoveL Offs(pOrigin,295.05,219.62,6.00),v60,z5,tPen\WObj:=wPaper;
    MoveL Offs(pOrigin,293.77,218.77,6.00),vTravel,z5,tPen\WObj:=wPaper;
    MoveL Offs(pOrigin,293.77,218.77,0.00),v60,z0,tPen\WObj:=wPaper;
    MoveL Offs(pOrigin,292.92,219.62,0.00),v40,z0,tPen\WObj:=wPaper;
    MoveL Offs(pOrigin,293.77,218.77,0.00),v40,fine,tPen\WObj:=wPaper;
  ENDPROC

  PROC DrawPart55()
    MoveL Offs(pOrigin,293.77,218.77,6.00),v60,z5,tPen\WObj:=wPaper;
    MoveL Offs(pOrigin,296.11,218.35,6.00),vTravel,z5,tPen\WObj:=wPaper;
    MoveL Offs(pOrigin,296.11,218.35,0.00),v60,z0,tPen\WObj:=wPaper;
    MoveL Offs(pOrigin,296.33,217.93,0.00),v40,z0,tPen\WObj:=wPaper;
    MoveL Offs(pOrigin,296.11,218.35,0.00),v40,z0,tPen\WObj:=wPaper;
    MoveL Offs(pOrigin,296.75,217.71,0.00),v40,z0,tPen\WObj:=wPaper;
    MoveL Offs(pOrigin,296.96,217.29,0.00),v40,z0,tPen\WObj:=wPaper;
    MoveL Offs(pOrigin,296.75,217.71,0.00),v40,z0,tPen\WObj:=wPaper;
    MoveL Offs(pOrigin,297.39,217.07,0.00),v40,z0,tPen\WObj:=wPaper;
    MoveL Offs(pOrigin,297.60,216.65,0.00),v40,z0,tPen\WObj:=wPaper;
    MoveL Offs(pOrigin,297.39,217.07,0.00),v40,z0,tPen\WObj:=wPaper;
    MoveL Offs(pOrigin,298.02,216.44,0.00),v40,z0,tPen\WObj:=wPaper;
    MoveL Offs(pOrigin,298.45,216.01,0.00),v40,z0,tPen\WObj:=wPaper;
    MoveL Offs(pOrigin,298.02,216.44,0.00),v40,z0,tPen\WObj:=wPaper;
    MoveL Offs(pOrigin,298.88,215.80,0.00),v40,z0,tPen\WObj:=wPaper;
    MoveL Offs(pOrigin,299.09,215.38,0.00),v40,z0,tPen\WObj:=wPaper;
    MoveL Offs(pOrigin,298.88,215.80,0.00),v40,fine,tPen\WObj:=wPaper;
    MoveL Offs(pOrigin,298.88,215.80,6.00),v60,z5,tPen\WObj:=wPaper;
    MoveL Offs(pOrigin,299.73,214.74,6.00),vTravel,z5,tPen\WObj:=wPaper;
    MoveL Offs(pOrigin,299.73,214.74,0.00),v60,z0,tPen\WObj:=wPaper;
    MoveL Offs(pOrigin,299.51,215.16,0.00),v40,z0,tPen\WObj:=wPaper;
    MoveL Offs(pOrigin,299.73,214.74,0.00),v40,z0,tPen\WObj:=wPaper;
    MoveL Offs(pOrigin,300.36,214.10,0.00),v40,z0,tPen\WObj:=wPaper;
    MoveL Offs(pOrigin,300.15,214.52,0.00),v40,z0,tPen\WObj:=wPaper;
    MoveL Offs(pOrigin,300.36,214.10,0.00),v40,fine,tPen\WObj:=wPaper;
    MoveL Offs(pOrigin,300.36,214.10,6.00),v60,z5,tPen\WObj:=wPaper;
    MoveL Offs(pOrigin,299.02,213.39,6.00),vTravel,z5,tPen\WObj:=wPaper;
    MoveL Offs(pOrigin,299.02,213.39,0.00),v60,z0,tPen\WObj:=wPaper;
    MoveL Offs(pOrigin,294.20,218.14,0.00),v40,z0,tPen\WObj:=wPaper;
    MoveL Offs(pOrigin,299.02,213.39,0.00),v40,fine,tPen\WObj:=wPaper;
    MoveL Offs(pOrigin,299.02,213.39,6.00),v60,z5,tPen\WObj:=wPaper;
    MoveL Offs(pOrigin,300.79,211.55,6.00),vTravel,z5,tPen\WObj:=wPaper;
    MoveL Offs(pOrigin,300.79,211.55,0.00),v60,z0,tPen\WObj:=wPaper;
    MoveL Offs(pOrigin,299.30,213.04,0.00),v40,z0,tPen\WObj:=wPaper;
    MoveL Offs(pOrigin,300.79,211.55,0.00),v40,z0,tPen\WObj:=wPaper;
    MoveL Offs(pOrigin,301.42,210.70,0.00),v40,z0,tPen\WObj:=wPaper;
    MoveL Offs(pOrigin,301.00,211.34,0.00),v40,z0,tPen\WObj:=wPaper;
    MoveL Offs(pOrigin,301.42,210.70,0.00),v40,fine,tPen\WObj:=wPaper;
    MoveL Offs(pOrigin,301.42,210.70,6.00),v60,z5,tPen\WObj:=wPaper;
    MoveL Offs(pOrigin,302.49,209.64,6.00),vTravel,z5,tPen\WObj:=wPaper;
    MoveL Offs(pOrigin,302.49,209.64,0.00),v60,z0,tPen\WObj:=wPaper;
    MoveL Offs(pOrigin,301.85,210.27,0.00),v40,z0,tPen\WObj:=wPaper;
    MoveL Offs(pOrigin,302.49,209.64,0.00),v40,fine,tPen\WObj:=wPaper;
    MoveL Offs(pOrigin,302.49,209.64,6.00),v60,z5,tPen\WObj:=wPaper;
    MoveL Offs(pOrigin,304.19,209.85,6.00),vTravel,z5,tPen\WObj:=wPaper;
    MoveL Offs(pOrigin,304.19,209.85,0.00),v60,z0,tPen\WObj:=wPaper;
    MoveL Offs(pOrigin,303.98,210.27,0.00),v40,z0,tPen\WObj:=wPaper;
    MoveL Offs(pOrigin,304.19,209.85,0.00),v40,z0,tPen\WObj:=wPaper;
    MoveL Offs(pOrigin,304.83,209.21,0.00),v40,z0,tPen\WObj:=wPaper;
    MoveL Offs(pOrigin,305.04,208.79,0.00),v40,z0,tPen\WObj:=wPaper;
    MoveL Offs(pOrigin,304.83,209.21,0.00),v40,fine,tPen\WObj:=wPaper;
    MoveL Offs(pOrigin,304.83,209.21,6.00),v60,z5,tPen\WObj:=wPaper;
    MoveL Offs(pOrigin,305.89,207.94,6.00),vTravel,z5,tPen\WObj:=wPaper;
    MoveL Offs(pOrigin,305.89,207.94,0.00),v60,z0,tPen\WObj:=wPaper;
    MoveL Offs(pOrigin,306.10,207.51,0.00),v40,z0,tPen\WObj:=wPaper;
    MoveL Offs(pOrigin,305.89,207.94,0.00),v40,z0,tPen\WObj:=wPaper;
    MoveL Offs(pOrigin,306.52,207.09,0.00),v40,z0,tPen\WObj:=wPaper;
    MoveL Offs(pOrigin,306.74,206.66,0.00),v40,z0,tPen\WObj:=wPaper;
    MoveL Offs(pOrigin,306.52,207.09,0.00),v40,fine,tPen\WObj:=wPaper;
    MoveL Offs(pOrigin,306.52,207.09,6.00),v60,z5,tPen\WObj:=wPaper;
    MoveL Offs(pOrigin,305.04,206.45,6.00),vTravel,z5,tPen\WObj:=wPaper;
    MoveL Offs(pOrigin,305.04,206.45,0.00),v60,z0,tPen\WObj:=wPaper;
    MoveL Offs(pOrigin,304.61,206.88,0.00),v40,z0,tPen\WObj:=wPaper;
    MoveL Offs(pOrigin,305.04,206.45,0.00),v40,z0,tPen\WObj:=wPaper;
    MoveL Offs(pOrigin,305.67,205.60,0.00),v40,z0,tPen\WObj:=wPaper;
    MoveL Offs(pOrigin,305.25,206.24,0.00),v40,z0,tPen\WObj:=wPaper;
    MoveL Offs(pOrigin,305.67,205.60,0.00),v40,fine,tPen\WObj:=wPaper;
    MoveL Offs(pOrigin,305.67,205.60,6.00),v60,z5,tPen\WObj:=wPaper;
    MoveL Offs(pOrigin,307.59,205.60,6.00),vTravel,z5,tPen\WObj:=wPaper;
    MoveL Offs(pOrigin,307.59,205.60,0.00),v60,z0,tPen\WObj:=wPaper;
    MoveL Offs(pOrigin,307.38,206.02,0.00),v40,z0,tPen\WObj:=wPaper;
    MoveL Offs(pOrigin,307.59,205.60,0.00),v40,fine,tPen\WObj:=wPaper;
    MoveL Offs(pOrigin,307.59,205.60,6.00),v60,z5,tPen\WObj:=wPaper;
    MoveL Offs(pOrigin,307.80,203.05,6.00),vTravel,z5,tPen\WObj:=wPaper;
    MoveL Offs(pOrigin,307.80,203.05,0.00),v60,z0,tPen\WObj:=wPaper;
    MoveL Offs(pOrigin,307.16,203.69,0.00),v40,z0,tPen\WObj:=wPaper;
    MoveL Offs(pOrigin,307.80,203.05,0.00),v40,fine,tPen\WObj:=wPaper;
    MoveL Offs(pOrigin,307.80,203.05,6.00),v60,z5,tPen\WObj:=wPaper;
    MoveL Offs(pOrigin,309.71,202.84,6.00),vTravel,z5,tPen\WObj:=wPaper;
    MoveL Offs(pOrigin,309.71,202.84,0.00),v60,z0,tPen\WObj:=wPaper;
    MoveL Offs(pOrigin,309.50,203.26,0.00),v40,z0,tPen\WObj:=wPaper;
    MoveL Offs(pOrigin,309.71,202.84,0.00),v40,z0,tPen\WObj:=wPaper;
    MoveL Offs(pOrigin,310.35,201.99,0.00),v40,z0,tPen\WObj:=wPaper;
    MoveL Offs(pOrigin,309.92,202.62,0.00),v40,z0,tPen\WObj:=wPaper;
    MoveL Offs(pOrigin,310.35,201.99,0.00),v40,fine,tPen\WObj:=wPaper;
    MoveL Offs(pOrigin,310.35,201.99,6.00),v60,z5,tPen\WObj:=wPaper;
    MoveL Offs(pOrigin,310.14,200.07,6.00),vTravel,z5,tPen\WObj:=wPaper;
    MoveL Offs(pOrigin,310.14,200.07,0.00),v60,z0,tPen\WObj:=wPaper;
    MoveL Offs(pOrigin,309.71,200.50,0.00),v40,z0,tPen\WObj:=wPaper;
    MoveL Offs(pOrigin,310.14,200.07,0.00),v40,fine,tPen\WObj:=wPaper;
    MoveL Offs(pOrigin,310.14,200.07,6.00),v60,z5,tPen\WObj:=wPaper;
    MoveL Offs(pOrigin,311.84,200.29,6.00),vTravel,z5,tPen\WObj:=wPaper;
    MoveL Offs(pOrigin,311.84,200.29,0.00),v60,z0,tPen\WObj:=wPaper;
    MoveL Offs(pOrigin,311.20,200.93,0.00),v40,z0,tPen\WObj:=wPaper;
    MoveL Offs(pOrigin,311.84,200.29,0.00),v40,fine,tPen\WObj:=wPaper;
    MoveL Offs(pOrigin,311.84,200.29,6.00),v60,z5,tPen\WObj:=wPaper;
    MoveL Offs(pOrigin,311.20,198.59,6.00),vTravel,z5,tPen\WObj:=wPaper;
    MoveL Offs(pOrigin,311.20,198.59,0.00),v60,z0,tPen\WObj:=wPaper;
    MoveL Offs(pOrigin,310.77,199.23,0.00),v40,z0,tPen\WObj:=wPaper;
    MoveL Offs(pOrigin,311.20,198.59,0.00),v40,fine,tPen\WObj:=wPaper;
    MoveL Offs(pOrigin,311.20,198.59,6.00),v60,z5,tPen\WObj:=wPaper;
    MoveL Offs(pOrigin,313.11,198.38,6.00),vTravel,z5,tPen\WObj:=wPaper;
    MoveL Offs(pOrigin,313.11,198.38,0.00),v60,z0,tPen\WObj:=wPaper;
    MoveL Offs(pOrigin,312.69,199.01,0.00),v40,z0,tPen\WObj:=wPaper;
    MoveL Offs(pOrigin,313.11,198.38,0.00),v40,fine,tPen\WObj:=wPaper;
    MoveL Offs(pOrigin,313.11,198.38,6.00),v60,z5,tPen\WObj:=wPaper;
    MoveL Offs(pOrigin,312.69,196.89,6.00),vTravel,z5,tPen\WObj:=wPaper;
    MoveL Offs(pOrigin,312.69,196.89,0.00),v60,z0,tPen\WObj:=wPaper;
    MoveL Offs(pOrigin,312.05,197.52,0.00),v40,z0,tPen\WObj:=wPaper;
    MoveL Offs(pOrigin,312.69,196.89,0.00),v40,z0,tPen\WObj:=wPaper;
    MoveL Offs(pOrigin,313.33,196.04,0.00),v40,z0,tPen\WObj:=wPaper;
    MoveL Offs(pOrigin,312.90,196.46,0.00),v40,z0,tPen\WObj:=wPaper;
    MoveL Offs(pOrigin,313.33,196.04,0.00),v40,fine,tPen\WObj:=wPaper;
    MoveL Offs(pOrigin,313.33,196.04,6.00),v60,z5,tPen\WObj:=wPaper;
    MoveL Offs(pOrigin,312.69,194.34,6.00),vTravel,z5,tPen\WObj:=wPaper;
    MoveL Offs(pOrigin,312.69,194.34,0.00),v60,z0,tPen\WObj:=wPaper;
    MoveL Offs(pOrigin,313.11,194.55,0.00),v40,z0,tPen\WObj:=wPaper;
    MoveL Offs(pOrigin,312.69,194.34,0.00),v40,z0,tPen\WObj:=wPaper;
    MoveL Offs(pOrigin,311.62,193.91,0.00),v40,z0,tPen\WObj:=wPaper;
    MoveL Offs(pOrigin,312.05,194.12,0.00),v40,z0,tPen\WObj:=wPaper;
  ENDPROC

  PROC DrawPart56()
    MoveL Offs(pOrigin,311.62,193.91,0.00),v40,fine,tPen\WObj:=wPaper;
    MoveL Offs(pOrigin,311.62,193.91,6.00),v60,z5,tPen\WObj:=wPaper;
    MoveL Offs(pOrigin,310.35,193.27,6.00),vTravel,z5,tPen\WObj:=wPaper;
    MoveL Offs(pOrigin,310.35,193.27,0.00),v60,z0,tPen\WObj:=wPaper;
    MoveL Offs(pOrigin,310.77,193.49,0.00),v40,z0,tPen\WObj:=wPaper;
    MoveL Offs(pOrigin,310.35,193.27,0.00),v40,fine,tPen\WObj:=wPaper;
    MoveL Offs(pOrigin,310.35,193.27,6.00),v60,z5,tPen\WObj:=wPaper;
    MoveL Offs(pOrigin,310.14,191.79,6.00),vTravel,z5,tPen\WObj:=wPaper;
    MoveL Offs(pOrigin,310.14,191.79,0.00),v60,z0,tPen\WObj:=wPaper;
    MoveL Offs(pOrigin,310.56,192.00,0.00),v40,z0,tPen\WObj:=wPaper;
    MoveL Offs(pOrigin,310.14,191.79,0.00),v40,fine,tPen\WObj:=wPaper;
    MoveL Offs(pOrigin,310.14,191.79,6.00),v60,z5,tPen\WObj:=wPaper;
    MoveL Offs(pOrigin,307.59,192.00,6.00),vTravel,z5,tPen\WObj:=wPaper;
    MoveL Offs(pOrigin,307.59,192.00,0.00),v60,z0,tPen\WObj:=wPaper;
    MoveL Offs(pOrigin,308.01,192.21,0.00),v40,z0,tPen\WObj:=wPaper;
    MoveL Offs(pOrigin,307.59,192.00,0.00),v40,fine,tPen\WObj:=wPaper;
    MoveL Offs(pOrigin,307.59,192.00,6.00),v60,z5,tPen\WObj:=wPaper;
    MoveL Offs(pOrigin,303.98,190.30,6.00),vTravel,z5,tPen\WObj:=wPaper;
    MoveL Offs(pOrigin,303.98,190.30,0.00),v60,z0,tPen\WObj:=wPaper;
    MoveL Offs(pOrigin,304.40,190.51,0.00),v40,z0,tPen\WObj:=wPaper;
    MoveL Offs(pOrigin,303.98,190.30,0.00),v40,fine,tPen\WObj:=wPaper;
    MoveL Offs(pOrigin,303.98,190.30,6.00),v60,z5,tPen\WObj:=wPaper;
    MoveL Offs(pOrigin,300.58,189.66,6.00),vTravel,z5,tPen\WObj:=wPaper;
    MoveL Offs(pOrigin,300.58,189.66,0.00),v60,z0,tPen\WObj:=wPaper;
    MoveL Offs(pOrigin,301.00,189.45,0.00),v40,z0,tPen\WObj:=wPaper;
    MoveL Offs(pOrigin,300.58,189.66,0.00),v40,fine,tPen\WObj:=wPaper;
    MoveL Offs(pOrigin,300.58,189.66,6.00),v60,z5,tPen\WObj:=wPaper;
    MoveL Offs(pOrigin,297.39,191.36,6.00),vTravel,z5,tPen\WObj:=wPaper;
    MoveL Offs(pOrigin,297.39,191.36,0.00),v60,z0,tPen\WObj:=wPaper;
    MoveL Offs(pOrigin,297.39,191.79,0.00),v40,z0,tPen\WObj:=wPaper;
    MoveL Offs(pOrigin,296.54,192.00,0.00),v40,z0,tPen\WObj:=wPaper;
    MoveL Offs(pOrigin,296.54,192.00,0.00),v40,z0,tPen\WObj:=wPaper;
    MoveL Offs(pOrigin,296.33,192.64,0.00),v40,z0,tPen\WObj:=wPaper;
    MoveL Offs(pOrigin,295.26,192.85,0.00),v40,z0,tPen\WObj:=wPaper;
    MoveL Offs(pOrigin,295.26,192.85,0.00),v40,z0,tPen\WObj:=wPaper;
    MoveL Offs(pOrigin,295.26,192.21,0.00),v40,z0,tPen\WObj:=wPaper;
    MoveL Offs(pOrigin,295.69,191.79,0.00),v40,z0,tPen\WObj:=wPaper;
    MoveL Offs(pOrigin,296.33,191.79,0.00),v40,z0,tPen\WObj:=wPaper;
    MoveL Offs(pOrigin,296.33,191.79,0.00),v40,z0,tPen\WObj:=wPaper;
    MoveL Offs(pOrigin,296.54,191.15,0.00),v40,z0,tPen\WObj:=wPaper;
    MoveL Offs(pOrigin,297.17,190.94,0.00),v40,fine,tPen\WObj:=wPaper;
    MoveL Offs(pOrigin,297.17,190.94,6.00),v60,z5,tPen\WObj:=wPaper;
    MoveL Offs(pOrigin,295.26,192.85,6.00),vTravel,z5,tPen\WObj:=wPaper;
    MoveL Offs(pOrigin,295.26,192.85,0.00),v60,z0,tPen\WObj:=wPaper;
    MoveL Offs(pOrigin,294.41,193.27,0.00),v40,z0,tPen\WObj:=wPaper;
    MoveL Offs(pOrigin,293.56,194.34,0.00),v40,z0,tPen\WObj:=wPaper;
    MoveL Offs(pOrigin,293.77,194.12,0.00),v40,fine,tPen\WObj:=wPaper;
    MoveL Offs(pOrigin,293.77,194.12,6.00),v60,z5,tPen\WObj:=wPaper;
    MoveL Offs(pOrigin,280.39,204.32,6.00),vTravel,z5,tPen\WObj:=wPaper;
    MoveL Offs(pOrigin,280.39,204.32,0.00),v60,z0,tPen\WObj:=wPaper;
    MoveL Offs(pOrigin,280.60,204.75,0.00),v40,z0,tPen\WObj:=wPaper;
    MoveL Offs(pOrigin,280.39,204.32,0.00),v40,z0,tPen\WObj:=wPaper;
    MoveL Offs(pOrigin,280.81,204.96,0.00),v40,z0,tPen\WObj:=wPaper;
    MoveL Offs(pOrigin,281.02,205.39,0.00),v40,z0,tPen\WObj:=wPaper;
    MoveL Offs(pOrigin,280.81,204.96,0.00),v40,z0,tPen\WObj:=wPaper;
    MoveL Offs(pOrigin,281.24,205.81,0.00),v40,z0,tPen\WObj:=wPaper;
    MoveL Offs(pOrigin,281.45,206.24,0.00),v40,z0,tPen\WObj:=wPaper;
    MoveL Offs(pOrigin,281.24,205.81,0.00),v40,fine,tPen\WObj:=wPaper;
    MoveL Offs(pOrigin,281.24,205.81,6.00),v60,z5,tPen\WObj:=wPaper;
    MoveL Offs(pOrigin,282.09,207.51,6.00),vTravel,z5,tPen\WObj:=wPaper;
    MoveL Offs(pOrigin,282.09,207.51,0.00),v60,z0,tPen\WObj:=wPaper;
    MoveL Offs(pOrigin,282.30,207.94,0.00),v40,z0,tPen\WObj:=wPaper;
    MoveL Offs(pOrigin,282.09,207.51,0.00),v40,z0,tPen\WObj:=wPaper;
    MoveL Offs(pOrigin,282.51,208.36,0.00),v40,z0,tPen\WObj:=wPaper;
    MoveL Offs(pOrigin,282.73,208.79,0.00),v40,z0,tPen\WObj:=wPaper;
    MoveL Offs(pOrigin,282.51,208.36,0.00),v40,fine,tPen\WObj:=wPaper;
    MoveL Offs(pOrigin,282.51,208.36,6.00),v60,z5,tPen\WObj:=wPaper;
    MoveL Offs(pOrigin,281.66,209.85,6.00),vTravel,z5,tPen\WObj:=wPaper;
    MoveL Offs(pOrigin,281.66,209.85,0.00),v60,z0,tPen\WObj:=wPaper;
    MoveL Offs(pOrigin,282.09,210.49,0.00),v40,z0,tPen\WObj:=wPaper;
    MoveL Offs(pOrigin,281.66,209.85,0.00),v40,fine,tPen\WObj:=wPaper;
    MoveL Offs(pOrigin,281.66,209.85,6.00),v60,z5,tPen\WObj:=wPaper;
    MoveL Offs(pOrigin,282.30,210.91,6.00),vTravel,z5,tPen\WObj:=wPaper;
    MoveL Offs(pOrigin,282.30,210.91,0.00),v60,z0,tPen\WObj:=wPaper;
    MoveL Offs(pOrigin,282.51,211.34,0.00),v40,z0,tPen\WObj:=wPaper;
    MoveL Offs(pOrigin,282.30,210.91,0.00),v40,fine,tPen\WObj:=wPaper;
    MoveL Offs(pOrigin,282.30,210.91,6.00),v60,z5,tPen\WObj:=wPaper;
    MoveL Offs(pOrigin,283.36,210.06,6.00),vTravel,z5,tPen\WObj:=wPaper;
    MoveL Offs(pOrigin,283.36,210.06,0.00),v60,z0,tPen\WObj:=wPaper;
    MoveL Offs(pOrigin,283.58,210.49,0.00),v40,z0,tPen\WObj:=wPaper;
    MoveL Offs(pOrigin,283.36,210.06,0.00),v40,fine,tPen\WObj:=wPaper;
    MoveL Offs(pOrigin,283.36,210.06,6.00),v60,z5,tPen\WObj:=wPaper;
    MoveL Offs(pOrigin,283.15,212.61,6.00),vTravel,z5,tPen\WObj:=wPaper;
    MoveL Offs(pOrigin,283.15,212.61,0.00),v60,z0,tPen\WObj:=wPaper;
    MoveL Offs(pOrigin,283.36,213.04,0.00),v40,z0,tPen\WObj:=wPaper;
    MoveL Offs(pOrigin,283.15,212.61,0.00),v40,fine,tPen\WObj:=wPaper;
    MoveL Offs(pOrigin,283.15,212.61,6.00),v60,z5,tPen\WObj:=wPaper;
    MoveL Offs(pOrigin,278.90,213.89,6.00),vTravel,z5,tPen\WObj:=wPaper;
    MoveL Offs(pOrigin,278.90,213.89,0.00),v60,z0,tPen\WObj:=wPaper;
    MoveL Offs(pOrigin,280.81,215.59,0.00),v40,z0,tPen\WObj:=wPaper;
    MoveL Offs(pOrigin,283.36,219.41,0.00),v40,fine,tPen\WObj:=wPaper;
    MoveL Offs(pOrigin,283.36,219.41,6.00),v60,z5,tPen\WObj:=wPaper;
    MoveL Offs(pOrigin,282.51,224.30,6.00),vTravel,z5,tPen\WObj:=wPaper;
    MoveL Offs(pOrigin,282.51,224.30,0.00),v60,z0,tPen\WObj:=wPaper;
    MoveL Offs(pOrigin,279.75,220.26,0.00),v40,z0,tPen\WObj:=wPaper;
    MoveL Offs(pOrigin,276.99,217.50,0.00),v40,z0,tPen\WObj:=wPaper;
    MoveL Offs(pOrigin,273.38,214.88,0.00),v40,z0,tPen\WObj:=wPaper;
    MoveL Offs(pOrigin,268.49,212.40,0.00),v40,fine,tPen\WObj:=wPaper;
    MoveL Offs(pOrigin,268.49,212.40,6.00),v60,z5,tPen\WObj:=wPaper;
    MoveL Offs(pOrigin,267.64,215.38,6.00),vTravel,z5,tPen\WObj:=wPaper;
    MoveL Offs(pOrigin,267.64,215.38,0.00),v60,z0,tPen\WObj:=wPaper;
    MoveL Offs(pOrigin,265.65,213.68,0.00),v40,z0,tPen\WObj:=wPaper;
    MoveL Offs(pOrigin,265.09,212.75,0.00),v40,z0,tPen\WObj:=wPaper;
    MoveL Offs(pOrigin,262.33,211.20,0.00),v40,z0,tPen\WObj:=wPaper;
    MoveL Offs(pOrigin,259.56,210.49,0.00),v40,z0,tPen\WObj:=wPaper;
    MoveL Offs(pOrigin,259.56,210.49,0.00),v40,z0,tPen\WObj:=wPaper;
    MoveL Offs(pOrigin,253.61,209.21,0.00),v40,z0,tPen\WObj:=wPaper;
    MoveL Offs(pOrigin,247.24,208.36,0.00),v40,z0,tPen\WObj:=wPaper;
    MoveL Offs(pOrigin,241.07,208.36,0.00),v40,z0,tPen\WObj:=wPaper;
    MoveL Offs(pOrigin,238.10,208.79,0.00),v40,z0,tPen\WObj:=wPaper;
    MoveL Offs(pOrigin,238.10,208.79,0.00),v40,z0,tPen\WObj:=wPaper;
    MoveL Offs(pOrigin,237.04,209.00,0.00),v40,z0,tPen\WObj:=wPaper;
    MoveL Offs(pOrigin,237.04,209.00,0.00),v40,z0,tPen\WObj:=wPaper;
    MoveL Offs(pOrigin,237.46,208.15,0.00),v40,z0,tPen\WObj:=wPaper;
    MoveL Offs(pOrigin,237.89,208.15,0.00),v40,z0,tPen\WObj:=wPaper;
    MoveL Offs(pOrigin,238.10,208.79,0.00),v40,z0,tPen\WObj:=wPaper;
    MoveL Offs(pOrigin,238.10,208.15,0.00),v40,z0,tPen\WObj:=wPaper;
    MoveL Offs(pOrigin,240.86,207.51,0.00),v40,z0,tPen\WObj:=wPaper;
    MoveL Offs(pOrigin,248.30,207.51,0.00),v40,z0,tPen\WObj:=wPaper;
    MoveL Offs(pOrigin,256.16,208.79,0.00),v40,z0,tPen\WObj:=wPaper;
  ENDPROC

